   1:  PR[91,3] = PR[90,3] + 57.179;
   1:L PR[91] R[100]mm/sec CNT100;
   1:  PR[91,1] = PR[90,1] + 0.045;
   1:  PR[91,2] = PR[90,2] + -22.058;
   1:  PR[91,3] = PR[90,3] + 57.186;
   1:L PR[91] R[100]mm/sec CNT100;
   1:  PR[91] = PR[90];
   1:  PR[91,1] = PR[90,1] + 1.559;
   1:  PR[91,2] = PR[90,2] + -22.487;
   1:  PR[91,3] = PR[90,3] + 58.520;
   1:L PR[91] R[100]mm/sec CNT100;
   1:  PR[91,1] = PR[90,1] + 2.758;
   1:  PR[91,2] = PR[90,2] + -22.482;
   1:  PR[91,3] = PR[90,3] + 57.203;
   1:L PR[91] R[100]mm/sec CNT100;
   1:  PR[91,1] = PR[90,1] + 3.956;
   1:  PR[91,2] = PR[90,2] + -22.416;
   1:  PR[91,3] = PR[90,3] + 57.213;
   1:L PR[91] R[100]mm/sec CNT100;
   1:  PR[91,1] = PR[90,1] + 5.149;
   1:  PR[91,2] = PR[90,2] + -22.289;
   1:  PR[91,3] = PR[90,3] + 57.223;
   1:L PR[91] R[100]mm/sec CNT100;
   1:  PR[91,1] = PR[90,1] + 6.334;
   1:  PR[91,2] = PR[90,2] + -22.101;
   1:  PR[91,3] = PR[90,3] + 57.234;
   1:L PR[91] R[100]mm/sec CNT100;
   1:  PR[91,1] = PR[90,1] + 7.176;
   1:  PR[91,2] = PR[90,2] + -21.924;
   1:  PR[91,3] = PR[90,3] + 57.244;
   1:L PR[91] R[100]mm/sec CNT100;
   1:  PR[91,1] = PR[90,1] + 7.504;
   1:  PR[91,2] = PR[90,2] + -21.853;
   1:  PR[91,3] = PR[90,3] + 57.252;
   1:L PR[91] R[100]mm/sec CNT100;
   1:  PR[91,1] = PR[90,1] + 8.663;
   1:  PR[91,2] = PR[90,2] + -21.545;
   1:  PR[91,3] = PR[90,3] + 57.255;
   1:L PR[91] R[100]mm/sec CNT100;
   1:  PR[91,1] = PR[90,1] + 9.802;
   1:  PR[91,2] = PR[90,2] + -21.178;
   1:  PR[91,3] = PR[90,3] + 57.265;
   1:L PR[91] R[100]mm/sec CNT100;
   1:  PR[91,1] = PR[90,1] + 10.920;
   1:  PR[91,2] = PR[90,2] + -20.755;
   1:  PR[91,3] = PR[90,3] + 57.275;
   1:L PR[91] R[100]mm/sec CNT100;
   1:  PR[91,1] = PR[90,1] + 12.013;
   1:  PR[91,2] = PR[90,2] + -20.275;
   1:  PR[91,3] = PR[90,3] + 57.286;
   1:L PR[91] R[100]mm/sec CNT100;
   1:  PR[91,1] = PR[90,1] + 13.080;
   1:  PR[91,2] = PR[90,2] + -19.740;
   1:  PR[91,3] = PR[90,3] + 57.296;
   1:L PR[91] R[100]mm/sec CNT100;
   1:  PR[91,1] = PR[90,1] + 14.117;
   1:  PR[91,2] = PR[90,2] + -19.152;
   1:  PR[91,3] = PR[90,3] + 57.306;
   1:L PR[91] R[100]mm/sec CNT100;
   1:  PR[91,1] = PR[90,1] + 14.721;
   1:  PR[91,2] = PR[90,2] + -18.769;
   1:  PR[91,3] = PR[90,3] + 57.317;
   1:L PR[91] R[100]mm/sec CNT100;
   1:  PR[91,1] = PR[90,1] + 15.120;
   1:  PR[91,2] = PR[90,2] + -18.514;
   1:  PR[91,3] = PR[90,3] + 57.323;
   1:L PR[91] R[100]mm/sec CNT100;
   1:  PR[91,1] = PR[90,1] + 16.090;
   1:  PR[91,2] = PR[90,2] + -17.825;
   1:  PR[91,3] = PR[90,3] + 57.327;
   1:L PR[91] R[100]mm/sec CNT100;
   1:  PR[91,1] = PR[90,1] + 17.021;
   1:  PR[91,2] = PR[90,2] + -17.088;
   1:  PR[91,3] = PR[90,3] + 57.337;
   1:L PR[91] R[100]mm/sec CNT100;
   1:  PR[91,1] = PR[90,1] + 17.913;
   1:  PR[91,2] = PR[90,2] + -16.306;
   1:  PR[91,3] = PR[90,3] + 57.348;
   1:L PR[91] R[100]mm/sec CNT100;
   1:  PR[91,1] = PR[90,1] + 18.761;
   1:  PR[91,2] = PR[90,2] + -15.480;
   1:  PR[91,3] = PR[90,3] + 57.358;
   1:L PR[91] R[100]mm/sec CNT100;
   1:  PR[91,1] = PR[90,1] + 19.566;
   1:  PR[91,2] = PR[90,2] + -14.612;
   1:  PR[91,3] = PR[90,3] + 57.368;
   1:L PR[91] R[100]mm/sec CNT100;
   1:  PR[91,1] = PR[90,1] + 20.324;
   1:  PR[91,2] = PR[90,2] + -13.706;
   1:  PR[91,3] = PR[90,3] + 57.378;
   1:L PR[91] R[100]mm/sec CNT100;
   1:  PR[91,1] = PR[90,1] + 21.034;
   1:  PR[91,2] = PR[90,2] + -12.762;
   1:  PR[91,3] = PR[90,3] + 57.389;
   1:L PR[91] R[100]mm/sec CNT100;
   1:  PR[91,1] = PR[90,1] + 21.694;
   1:  PR[91,2] = PR[90,2] + -11.785;
   1:  PR[91,3] = PR[90,3] + 57.399;
   1:L PR[91] R[100]mm/sec CNT100;
   1:  PR[91,1] = PR[90,1] + 22.301;
   1:  PR[91,2] = PR[90,2] + -10.776;
   1:  PR[91,3] = PR[90,3] + 57.409;
   1:L PR[91] R[100]mm/sec CNT100;
   1:  PR[91,1] = PR[90,1] + 22.856;
   1:  PR[91,2] = PR[90,2] + -9.738;
   1:  PR[91,3] = PR[90,3] + 57.419;
   1:L PR[91] R[100]mm/sec CNT100;
   1:  PR[91,1] = PR[90,1] + 23.356;
   1:  PR[91,2] = PR[90,2] + -8.675;
   1:  PR[91,3] = PR[90,3] + 57.429;
   1:L PR[91] R[100]mm/sec CNT100;
   1:  PR[91,1] = PR[90,1] + 23.800;
   1:  PR[91,2] = PR[90,2] + -7.590;
   1:  PR[91,3] = PR[90,3] + 57.440;
   1:L PR[91] R[100]mm/sec CNT100;
   1:  PR[91,1] = PR[90,1] + 24.187;
   1:  PR[91,2] = PR[90,2] + -6.485;
   1:  PR[91,3] = PR[90,3] + 57.450;
   1:L PR[91] R[100]mm/sec CNT100;
   1:  PR[91,1] = PR[90,1] + 24.516;
   1:  PR[91,2] = PR[90,2] + -5.362;
   1:  PR[91,3] = PR[90,3] + 57.460;
   1:L PR[91] R[100]mm/sec CNT100;
   1:  PR[91,1] = PR[90,1] + 24.786;
   1:  PR[91,2] = PR[90,2] + -4.225;
   1:  PR[91,3] = PR[90,3] + 57.470;
   1:L PR[91] R[100]mm/sec CNT100;
   1:  PR[91,1] = PR[90,1] + 24.997;
   1:  PR[91,2] = PR[90,2] + -3.075;
   1:  PR[91,3] = PR[90,3] + 57.480;
   1:L PR[91] R[100]mm/sec CNT100;
   1:  PR[91,1] = PR[90,1] + 25.148;
   1:  PR[91,2] = PR[90,2] + -1.915;
   1:  PR[91,3] = PR[90,3] + 57.490;
   1:L PR[91] R[100]mm/sec CNT100;
   1:  PR[91,1] = PR[90,1] + 25.238;
   1:  PR[91,2] = PR[90,2] + -0.746;
   1:  PR[91,3] = PR[90,3] + 57.500;
   1:L PR[91] R[100]mm/sec CNT100;
   1:  PR[91,1] = PR[90,1] + 25.269;
   1:  PR[91,2] = PR[90,2] + 0.428;
   1:  PR[91,3] = PR[90,3] + 57.510;
   1:L PR[91] R[100]mm/sec CNT100;
   1:  PR[91,1] = PR[90,1] + 25.238;
   1:  PR[91,2] = PR[90,2] + 1.601;
   1:  PR[91,3] = PR[90,3] + 57.521;
   1:L PR[91] R[100]mm/sec CNT100;
   1:  PR[91,1] = PR[90,1] + 25.148;
   1:  PR[91,2] = PR[90,2] + 2.770;
   1:  PR[91,3] = PR[90,3] + 57.531;
   1:L PR[91] R[100]mm/sec CNT100;
   1:  PR[91,1] = PR[90,1] + 24.997;
   1:  PR[91,2] = PR[90,2] + 3.930;
   1:  PR[91,3] = PR[90,3] + 57.541;
   1:L PR[91] R[100]mm/sec CNT100;
   1:  PR[91,1] = PR[90,1] + 24.786;
   1:  PR[91,2] = PR[90,2] + 5.080;
   1:  PR[91,3] = PR[90,3] + 57.551;
   1:L PR[91] R[100]mm/sec CNT100;
   1:  PR[91,1] = PR[90,1] + 24.516;
   1:  PR[91,2] = PR[90,2] + 6.217;
   1:  PR[91,3] = PR[90,3] + 57.561;
   1:L PR[91] R[100]mm/sec CNT100;
   1:  PR[91,1] = PR[90,1] + 24.187;
   1:  PR[91,2] = PR[90,2] + 7.339;
   1:  PR[91,3] = PR[90,3] + 57.571;
   1:L PR[91] R[100]mm/sec CNT100;
   1:  PR[91,1] = PR[90,1] + 23.800;
   1:  PR[91,2] = PR[90,2] + 8.445;
   1:  PR[91,3] = PR[90,3] + 57.581;
   1:L PR[91] R[100]mm/sec CNT100;
   1:  PR[91,1] = PR[90,1] + 23.356;
   1:  PR[91,2] = PR[90,2] + 9.530;
   1:  PR[91,3] = PR[90,3] + 57.592;
   1:L PR[91] R[100]mm/sec CNT100;
   1:  PR[91,1] = PR[90,1] + 22.856;
   1:  PR[91,2] = PR[90,2] + 10.593;
   1:  PR[91,3] = PR[90,3] + 57.602;
   1:L PR[91] R[100]mm/sec CNT100;
   1:  PR[91,1] = PR[90,1] + 22.302;
   1:  PR[91,2] = PR[90,2] + 11.630;
   1:  PR[91,3] = PR[90,3] + 57.612;
   1:L PR[91] R[100]mm/sec CNT100;
   1:  PR[91,1] = PR[90,1] + 21.694;
   1:  PR[91,2] = PR[90,2] + 12.639;
   1:  PR[91,3] = PR[90,3] + 57.622;
   1:L PR[91] R[100]mm/sec CNT100;
   1:  PR[91,1] = PR[90,1] + 21.034;
   1:  PR[91,2] = PR[90,2] + 13.617;
   1:  PR[91,3] = PR[90,3] + 57.632;
   1:L PR[91] R[100]mm/sec CNT100;
   1:  PR[91,1] = PR[90,1] + 20.325;
   1:  PR[91,2] = PR[90,2] + 14.560;
   1:  PR[91,3] = PR[90,3] + 57.642;
   1:L PR[91] R[100]mm/sec CNT100;
   1:  PR[91,1] = PR[90,1] + 19.567;
   1:  PR[91,2] = PR[90,2] + 15.467;
   1:  PR[91,3] = PR[90,3] + 57.653;
   1:L PR[91] R[100]mm/sec CNT100;
   1:  PR[91,1] = PR[90,1] + 18.762;
   1:  PR[91,2] = PR[90,2] + 16.335;
   1:  PR[91,3] = PR[90,3] + 57.663;
   1:L PR[91] R[100]mm/sec CNT100;
   1:  PR[91,1] = PR[90,1] + 17.913;
   1:  PR[91,2] = PR[90,2] + 17.161;
   1:  PR[91,3] = PR[90,3] + 57.673;
   1:L PR[91] R[100]mm/sec CNT100;
   1:  PR[91,1] = PR[90,1] + 17.021;
   1:  PR[91,2] = PR[90,2] + 17.943;
   1:  PR[91,3] = PR[90,3] + 57.683;
   1:L PR[91] R[100]mm/sec CNT100;
   1:  PR[91,1] = PR[90,1] + 16.090;
   1:  PR[91,2] = PR[90,2] + 18.680;
   1:  PR[91,3] = PR[90,3] + 57.694;
   1:L PR[91] R[100]mm/sec CNT100;
   1:  PR[91,1] = PR[90,1] + 15.121;
   1:  PR[91,2] = PR[90,2] + 19.369;
   1:  PR[91,3] = PR[90,3] + 57.704;
   1:L PR[91] R[100]mm/sec CNT100;
   1:  PR[91,1] = PR[90,1] + 14.117;
   1:  PR[91,2] = PR[90,2] + 20.008;
   1:  PR[91,3] = PR[90,3] + 57.714;
   1:L PR[91] R[100]mm/sec CNT100;
   1:  PR[91,1] = PR[90,1] + 13.080;
   1:  PR[91,2] = PR[90,2] + 20.595;
   1:  PR[91,3] = PR[90,3] + 57.725;
   1:L PR[91] R[100]mm/sec CNT100;
   1:  PR[91,1] = PR[90,1] + 12.013;
   1:  PR[91,2] = PR[90,2] + 21.130;
   1:  PR[91,3] = PR[90,3] + 57.735;
   1:L PR[91] R[100]mm/sec CNT100;
   1:  PR[91,1] = PR[90,1] + 10.919;
   1:  PR[91,2] = PR[90,2] + 21.610;
   1:  PR[91,3] = PR[90,3] + 57.745;
   1:L PR[91] R[100]mm/sec CNT100;
   1:  PR[91,1] = PR[90,1] + 9.802;
   1:  PR[91,2] = PR[90,2] + 22.033;
   1:  PR[91,3] = PR[90,3] + 57.756;
   1:L PR[91] R[100]mm/sec CNT100;
   1:  PR[91,1] = PR[90,1] + 8.662;
   1:  PR[91,2] = PR[90,2] + 22.400;
   1:  PR[91,3] = PR[90,3] + 57.766;
   1:L PR[91] R[100]mm/sec CNT100;
   1:  PR[91,1] = PR[90,1] + 7.503;
   1:  PR[91,2] = PR[90,2] + 22.708;
   1:  PR[91,3] = PR[90,3] + 57.776;
   1:L PR[91] R[100]mm/sec CNT100;
   1:  PR[91,1] = PR[90,1] + 7.175;
   1:  PR[91,2] = PR[90,2] + 22.780;
   1:  PR[91,3] = PR[90,3] + 57.787;
   1:L PR[91] R[100]mm/sec CNT100;
   1:  PR[91,1] = PR[90,1] + 6.333;
   1:  PR[91,2] = PR[90,2] + 22.956;
   1:  PR[91,3] = PR[90,3] + 57.790;
   1:L PR[91] R[100]mm/sec CNT100;
   1:  PR[91,1] = PR[90,1] + 5.148;
   1:  PR[91,2] = PR[90,2] + 23.144;
   1:  PR[91,3] = PR[90,3] + 57.797;
   1:L PR[91] R[100]mm/sec CNT100;
   1:  PR[91,1] = PR[90,1] + 3.955;
   1:  PR[91,2] = PR[90,2] + 23.271;
   1:  PR[91,3] = PR[90,3] + 57.807;
   1:L PR[91] R[100]mm/sec CNT100;
   1:  PR[91,1] = PR[90,1] + 2.757;
   1:  PR[91,2] = PR[90,2] + 23.337;
   1:  PR[91,3] = PR[90,3] + 57.818;
   1:L PR[91] R[100]mm/sec CNT100;
   1:  PR[91,1] = PR[90,1] + 1.557;
   1:  PR[91,2] = PR[90,2] + 23.342;
   1:  PR[91,3] = PR[90,3] + 57.828;
   1:L PR[91] R[100]mm/sec CNT100;
   1:  PR[91,1] = PR[90,1] + 0.088;
   1:  PR[91,2] = PR[90,2] + 23.262;
   1:  PR[91,3] = PR[90,3] + 57.839;
   1:L PR[91] R[100]mm/sec CNT100;
   1:  PR[91,1] = PR[90,1] + -0.337;
   1:  PR[91,3] = PR[90,3] + 57.851;
   1:L PR[91] R[100]mm/sec CNT100;
   1:  PR[91,1] = PR[90,1] + -1.797;
   1:  PR[91,2] = PR[90,2] + 23.342;
   1:  PR[91,3] = PR[90,3] + 57.855;
   1:L PR[91] R[100]mm/sec CNT100;
   1:  PR[91,1] = PR[90,1] + -2.726;
   1:  PR[91,2] = PR[90,2] + 23.340;
   1:  PR[91,3] = PR[90,3] + 57.868;
   1:L PR[91] R[100]mm/sec CNT100;
   1:  PR[91,1] = PR[90,1] + -4.196;
   1:  PR[91,2] = PR[90,2] + 23.271;
   1:  PR[91,3] = PR[90,3] + 57.876;
   1:L PR[91] R[100]mm/sec CNT100;
   1:  PR[91,1] = PR[90,1] + -5.387;
   1:  PR[91,2] = PR[90,2] + 23.144;
   1:  PR[91,3] = PR[90,3] + 57.888;
   1:L PR[91] R[100]mm/sec CNT100;
   1:  PR[91,1] = PR[90,1] + -6.572;
   1:  PR[91,2] = PR[90,2] + 22.956;
   1:  PR[91,3] = PR[90,3] + 57.899;
   1:L PR[91] R[100]mm/sec CNT100;
   1:  PR[91,1] = PR[90,1] + -7.413;
   1:  PR[91,2] = PR[90,2] + 22.780;
   1:  PR[91,3] = PR[90,3] + 57.909;
   1:L PR[91] R[100]mm/sec CNT100;
   1:  PR[91,1] = PR[90,1] + -7.742;
   1:  PR[91,2] = PR[90,2] + 22.708;
   1:  PR[91,3] = PR[90,3] + 57.917;
   1:L PR[91] R[100]mm/sec CNT100;
   1:  PR[91,1] = PR[90,1] + -8.901;
   1:  PR[91,2] = PR[90,2] + 22.400;
   1:  PR[91,3] = PR[90,3] + 57.920;
   1:L PR[91] R[100]mm/sec CNT100;
   1:  PR[91,1] = PR[90,1] + -10.040;
   1:  PR[91,2] = PR[90,2] + 22.034;
   1:  PR[91,3] = PR[90,3] + 57.930;
   1:L PR[91] R[100]mm/sec CNT100;
   1:  PR[91,1] = PR[90,1] + -11.158;
   1:  PR[91,2] = PR[90,2] + 21.610;
   1:  PR[91,3] = PR[90,3] + 57.940;
   1:L PR[91] R[100]mm/sec CNT100;
   1:  PR[91,1] = PR[90,1] + -12.251;
   1:  PR[91,2] = PR[90,2] + 21.130;
   1:  PR[91,3] = PR[90,3] + 57.951;
   1:L PR[91] R[100]mm/sec CNT100;
   1:  PR[91,1] = PR[90,1] + -13.318;
   1:  PR[91,2] = PR[90,2] + 20.595;
   1:  PR[91,3] = PR[90,3] + 57.961;
   1:L PR[91] R[100]mm/sec CNT100;
   1:  PR[91,1] = PR[90,1] + -14.355;
   1:  PR[91,2] = PR[90,2] + 20.008;
   1:  PR[91,3] = PR[90,3] + 57.971;
   1:L PR[91] R[100]mm/sec CNT100;
   1:  PR[91,1] = PR[90,1] + -15.359;
   1:  PR[91,2] = PR[90,2] + 19.368;
   1:  PR[91,3] = PR[90,3] + 57.982;
   1:L PR[91] R[100]mm/sec CNT100;
   1:  PR[91,1] = PR[90,1] + -16.329;
   1:  PR[91,2] = PR[90,2] + 18.679;
   1:  PR[91,3] = PR[90,3] + 57.992;
   1:L PR[91] R[100]mm/sec CNT100;
   1:  PR[91,1] = PR[90,1] + -17.260;
   1:  PR[91,2] = PR[90,2] + 17.943;
   1:  PR[91,3] = PR[90,3] + 58.002;
   1:L PR[91] R[100]mm/sec CNT100;
   1:  PR[91,1] = PR[90,1] + -18.151;
   1:  PR[91,2] = PR[90,2] + 17.161;
   1:  PR[91,3] = PR[90,3] + 58.013;
   1:L PR[91] R[100]mm/sec CNT100;
   1:  PR[91,1] = PR[90,1] + -19.000;
   1:  PR[91,2] = PR[90,2] + 16.335;
   1:  PR[91,3] = PR[90,3] + 58.023;
   1:L PR[91] R[100]mm/sec CNT100;
   1:  PR[91,1] = PR[90,1] + -19.805;
   1:  PR[91,2] = PR[90,2] + 15.467;
   1:  PR[91,3] = PR[90,3] + 58.033;
   1:L PR[91] R[100]mm/sec CNT100;
   1:  PR[91,1] = PR[90,1] + -20.563;
   1:  PR[91,2] = PR[90,2] + 14.561;
   1:  PR[91,3] = PR[90,3] + 58.043;
   1:L PR[91] R[100]mm/sec CNT100;
   1:  PR[91,1] = PR[90,1] + -21.273;
   1:  PR[91,2] = PR[90,2] + 13.618;
   1:  PR[91,3] = PR[90,3] + 58.054;
   1:L PR[91] R[100]mm/sec CNT100;
   1:  PR[91,1] = PR[90,1] + -21.933;
   1:  PR[91,2] = PR[90,2] + 12.640;
   1:  PR[91,3] = PR[90,3] + 58.064;
   1:L PR[91] R[100]mm/sec CNT100;
   1:  PR[91,1] = PR[90,1] + -22.540;
   1:  PR[91,2] = PR[90,2] + 11.631;
   1:  PR[91,3] = PR[90,3] + 58.074;
   1:L PR[91] R[100]mm/sec CNT100;
   1:  PR[91,1] = PR[90,1] + -23.095;
   1:  PR[91,2] = PR[90,2] + 10.593;
   1:  PR[91,3] = PR[90,3] + 58.084;
   1:L PR[91] R[100]mm/sec CNT100;
   1:  PR[91,1] = PR[90,1] + -23.594;
   1:  PR[91,2] = PR[90,2] + 9.530;
   1:  PR[91,3] = PR[90,3] + 58.094;
   1:L PR[91] R[100]mm/sec CNT100;
   1:  PR[91,1] = PR[90,1] + -24.038;
   1:  PR[91,2] = PR[90,2] + 8.444;
   1:  PR[91,3] = PR[90,3] + 58.105;
   1:L PR[91] R[100]mm/sec CNT100;
   1:  PR[91,1] = PR[90,1] + -24.425;
   1:  PR[91,2] = PR[90,2] + 7.338;
   1:  PR[91,3] = PR[90,3] + 58.115;
   1:L PR[91] R[100]mm/sec CNT100;
   1:  PR[91,1] = PR[90,1] + -24.754;
   1:  PR[91,2] = PR[90,2] + 6.215;
   1:  PR[91,3] = PR[90,3] + 58.125;
   1:L PR[91] R[100]mm/sec CNT100;
   1:  PR[91,1] = PR[90,1] + -25.024;
   1:  PR[91,2] = PR[90,2] + 5.078;
   1:  PR[91,3] = PR[90,3] + 58.135;
   1:L PR[91] R[100]mm/sec CNT100;
   1:  PR[91,1] = PR[90,1] + -25.235;
   1:  PR[91,2] = PR[90,2] + 3.929;
   1:  PR[91,3] = PR[90,3] + 58.145;
   1:L PR[91] R[100]mm/sec CNT100;
   1:  PR[91,1] = PR[90,1] + -25.386;
   1:  PR[91,2] = PR[90,2] + 2.769;
   1:  PR[91,3] = PR[90,3] + 58.155;
   1:L PR[91] R[100]mm/sec CNT100;
   1:  PR[91,1] = PR[90,1] + -25.477;
   1:  PR[91,2] = PR[90,2] + 1.601;
   1:  PR[91,3] = PR[90,3] + 58.165;
   1:L PR[91] R[100]mm/sec CNT100;
   1:  PR[91,1] = PR[90,1] + -25.507;
   1:  PR[91,2] = PR[90,2] + 0.428;
   1:  PR[91,3] = PR[90,3] + 58.175;
   1:L PR[91] R[100]mm/sec CNT100;
   1:  PR[91,1] = PR[90,1] + -25.477;
   1:  PR[91,2] = PR[90,2] + -0.746;
   1:  PR[91,3] = PR[90,3] + 58.186;
   1:L PR[91] R[100]mm/sec CNT100;
   1:  PR[91,1] = PR[90,1] + -25.386;
   1:  PR[91,2] = PR[90,2] + -1.914;
   1:  PR[91,3] = PR[90,3] + 58.196;
   1:L PR[91] R[100]mm/sec CNT100;
   1:  PR[91,1] = PR[90,1] + -25.235;
   1:  PR[91,2] = PR[90,2] + -3.074;
   1:  PR[91,3] = PR[90,3] + 58.206;
   1:L PR[91] R[100]mm/sec CNT100;
   1:  PR[91,1] = PR[90,1] + -25.024;
   1:  PR[91,2] = PR[90,2] + -4.223;
   1:  PR[91,3] = PR[90,3] + 58.216;
   1:L PR[91] R[100]mm/sec CNT100;
   1:  PR[91,1] = PR[90,1] + -24.754;
   1:  PR[91,2] = PR[90,2] + -5.361;
   1:  PR[91,3] = PR[90,3] + 58.226;
   1:L PR[91] R[100]mm/sec CNT100;
   1:  PR[91,1] = PR[90,1] + -24.425;
   1:  PR[91,2] = PR[90,2] + -6.483;
   1:  PR[91,3] = PR[90,3] + 58.236;
   1:L PR[91] R[100]mm/sec CNT100;
   1:  PR[91,1] = PR[90,1] + -24.038;
   1:  PR[91,2] = PR[90,2] + -7.589;
   1:  PR[91,3] = PR[90,3] + 58.246;
   1:L PR[91] R[100]mm/sec CNT100;
   1:  PR[91,1] = PR[90,1] + -23.594;
   1:  PR[91,2] = PR[90,2] + -8.675;
   1:  PR[91,3] = PR[90,3] + 58.257;
   1:L PR[91] R[100]mm/sec CNT100;
   1:  PR[91,1] = PR[90,1] + -23.094;
   1:  PR[91,2] = PR[90,2] + -9.739;
   1:  PR[91,3] = PR[90,3] + 58.267;
   1:L PR[91] R[100]mm/sec CNT100;
   1:  PR[91,1] = PR[90,1] + -22.540;
   1:  PR[91,2] = PR[90,2] + -10.776;
   1:  PR[91,3] = PR[90,3] + 58.277;
   1:L PR[91] R[100]mm/sec CNT100;
   1:  PR[91,1] = PR[90,1] + -21.932;
   1:  PR[91,2] = PR[90,2] + -11.786;
   1:  PR[91,3] = PR[90,3] + 58.287;
   1:L PR[91] R[100]mm/sec CNT100;
   1:  PR[91,1] = PR[90,1] + -21.273;
   1:  PR[91,2] = PR[90,2] + -12.763;
   1:  PR[91,3] = PR[90,3] + 58.297;
   1:L PR[91] R[100]mm/sec CNT100;
   1:  PR[91,1] = PR[90,1] + -20.563;
   1:  PR[91,2] = PR[90,2] + -13.706;
   1:  PR[91,3] = PR[90,3] + 58.307;
   1:L PR[91] R[100]mm/sec CNT100;
   1:  PR[91,1] = PR[90,1] + -19.805;
   1:  PR[91,2] = PR[90,2] + -14.613;
   1:  PR[91,3] = PR[90,3] + 58.318;
   1:L PR[91] R[100]mm/sec CNT100;
   1:  PR[91,1] = PR[90,1] + -19.000;
   1:  PR[91,2] = PR[90,2] + -15.480;
   1:  PR[91,3] = PR[90,3] + 58.328;
   1:L PR[91] R[100]mm/sec CNT100;
   1:  PR[91,1] = PR[90,1] + -18.151;
   1:  PR[91,2] = PR[90,2] + -16.306;
   1:  PR[91,3] = PR[90,3] + 58.338;
   1:L PR[91] R[100]mm/sec CNT100;
   1:  PR[91,1] = PR[90,1] + -17.260;
   1:  PR[91,2] = PR[90,2] + -17.088;
   1:  PR[91,3] = PR[90,3] + 58.348;
   1:L PR[91] R[100]mm/sec CNT100;
   1:  PR[91,1] = PR[90,1] + -16.328;
   1:  PR[91,2] = PR[90,2] + -17.824;
   1:  PR[91,3] = PR[90,3] + 58.359;
   1:L PR[91] R[100]mm/sec CNT100;
   1:  PR[91,1] = PR[90,1] + -15.359;
   1:  PR[91,2] = PR[90,2] + -18.513;
   1:  PR[91,3] = PR[90,3] + 58.369;
   1:L PR[91] R[100]mm/sec CNT100;
   1:  PR[91,1] = PR[90,1] + -14.355;
   1:  PR[91,2] = PR[90,2] + -19.153;
   1:  PR[91,3] = PR[90,3] + 58.379;
   1:L PR[91] R[100]mm/sec CNT100;
   1:  PR[91,1] = PR[90,1] + -13.318;
   1:  PR[91,2] = PR[90,2] + -19.740;
   1:  PR[91,3] = PR[90,3] + 58.390;
   1:L PR[91] R[100]mm/sec CNT100;
   1:  PR[91,1] = PR[90,1] + -12.252;
   1:  PR[91,2] = PR[90,2] + -20.275;
   1:  PR[91,3] = PR[90,3] + 58.400;
   1:L PR[91] R[100]mm/sec CNT100;
   1:  PR[91,1] = PR[90,1] + -11.158;
   1:  PR[91,2] = PR[90,2] + -20.755;
   1:  PR[91,3] = PR[90,3] + 58.410;
   1:L PR[91] R[100]mm/sec CNT100;
   1:  PR[91,1] = PR[90,1] + -10.039;
   1:  PR[91,2] = PR[90,2] + -21.179;
   1:  PR[91,3] = PR[90,3] + 58.421;
   1:L PR[91] R[100]mm/sec CNT100;
   1:  PR[91,1] = PR[90,1] + -9.682;
   1:  PR[91,2] = PR[90,2] + -21.295;
   1:  PR[91,3] = PR[90,3] + 58.431;
   1:L PR[91] R[100]mm/sec CNT100;
   1:  PR[91,1] = PR[90,1] + -8.902;
   1:  PR[91,2] = PR[90,2] + -21.544;
   1:  PR[91,3] = PR[90,3] + 58.434;
   1:L PR[91] R[100]mm/sec CNT100;
   1:  PR[91,1] = PR[90,1] + -7.744;
   1:  PR[91,2] = PR[90,2] + -21.852;
   1:  PR[91,3] = PR[90,3] + 58.441;
   1:L PR[91] R[100]mm/sec CNT100;
   1:  PR[91,1] = PR[90,1] + -6.572;
   1:  PR[91,2] = PR[90,2] + -22.101;
   1:  PR[91,3] = PR[90,3] + 58.452;
   1:L PR[91] R[100]mm/sec CNT100;
   1:  PR[91,1] = PR[90,1] + -5.388;
   1:  PR[91,2] = PR[90,2] + -22.289;
   1:  PR[91,3] = PR[90,3] + 58.462;
   1:L PR[91] R[100]mm/sec CNT100;
   1:  PR[91,1] = PR[90,1] + -4.197;
   1:  PR[91,2] = PR[90,2] + -22.416;
   1:  PR[91,3] = PR[90,3] + 58.472;
   1:L PR[91] R[100]mm/sec CNT100;
   1:  PR[91,1] = PR[90,1] + -2.727;
   1:  PR[91,2] = PR[90,2] + -22.485;
   1:  PR[91,3] = PR[90,3] + 58.483;
   1:L PR[91] R[100]mm/sec CNT100;
   1:  PR[91,1] = PR[90,1] + -1.798;
   1:  PR[91,2] = PR[90,2] + -22.487;
   1:  PR[91,3] = PR[90,3] + 58.496;
   1:L PR[91] R[100]mm/sec CNT100;
   1:  PR[91,1] = PR[90,1] + -0.337;
   1:  PR[91,2] = PR[90,2] + -22.407;
   1:  PR[91,3] = PR[90,3] + 58.504;
   1:L PR[91] R[100]mm/sec CNT100;
   1:  PR[91,1] = PR[90,1] + 0.098;
   1:  PR[91,3] = PR[90,3] + 58.516;
   1:L PR[91] R[100]mm/sec CNT100;
   1:  PR[91] = PR[90];
   1:  PR[91,1] = PR[90,1] + 0.946;
   1:  PR[91,2] = PR[90,2] + -22.790;
   1:  PR[91,3] = PR[90,3] + 59.850;
   1:L PR[91] R[100]mm/sec CNT100;
   1:  PR[91,1] = PR[90,1] + 2.164;
   1:  PR[91,2] = PR[90,2] + -22.792;
   1:  PR[91,3] = PR[90,3] + 58.528;
   1:L PR[91] R[100]mm/sec CNT100;
   1:  PR[91,1] = PR[90,1] + 3.379;
   1:  PR[91,2] = PR[90,2] + -22.731;
   1:  PR[91,3] = PR[90,3] + 58.538;
   1:L PR[91] R[100]mm/sec CNT100;
   1:  PR[91,1] = PR[90,1] + 4.589;
   1:  PR[91,2] = PR[90,2] + -22.607;
   1:  PR[91,3] = PR[90,3] + 58.549;
   1:L PR[91] R[100]mm/sec CNT100;
   1:  PR[91,1] = PR[90,1] + 5.790;
   1:  PR[91,2] = PR[90,2] + -22.422;
   1:  PR[91,3] = PR[90,3] + 58.559;
   1:L PR[91] R[100]mm/sec CNT100;
   1:  PR[91,1] = PR[90,1] + 6.979;
   1:  PR[91,2] = PR[90,2] + -22.175;
   1:  PR[91,3] = PR[90,3] + 58.570;
   1:L PR[91] R[100]mm/sec CNT100;
   1:  PR[91,1] = PR[90,1] + 8.153;
   1:  PR[91,2] = PR[90,2] + -21.867;
   1:  PR[91,3] = PR[90,3] + 58.580;
   1:L PR[91] R[100]mm/sec CNT100;
   1:  PR[91,1] = PR[90,1] + 9.308;
   1:  PR[91,2] = PR[90,2] + -21.500;
   1:  PR[91,3] = PR[90,3] + 58.591;
   1:L PR[91] R[100]mm/sec CNT100;
   1:  PR[91,1] = PR[90,1] + 10.625;
   1:  PR[91,2] = PR[90,2] + -20.997;
   1:  PR[91,3] = PR[90,3] + 58.602;
   1:L PR[91] R[100]mm/sec CNT100;
   1:  PR[91,1] = PR[90,1] + 11.554;
   1:  PR[91,2] = PR[90,2] + -20.591;
   1:  PR[91,3] = PR[90,3] + 58.614;
   1:L PR[91] R[100]mm/sec CNT100;
   1:  PR[91,1] = PR[90,1] + 12.638;
   1:  PR[91,2] = PR[90,2] + -20.051;
   1:  PR[91,3] = PR[90,3] + 58.623;
   1:L PR[91] R[100]mm/sec CNT100;
   1:  PR[91,1] = PR[90,1] + 13.691;
   1:  PR[91,2] = PR[90,2] + -19.458;
   1:  PR[91,3] = PR[90,3] + 58.633;
   1:L PR[91] R[100]mm/sec CNT100;
   1:  PR[91,1] = PR[90,1] + 14.711;
   1:  PR[91,2] = PR[90,2] + -18.812;
   1:  PR[91,3] = PR[90,3] + 58.643;
   1:L PR[91] R[100]mm/sec CNT100;
   1:  PR[91,1] = PR[90,1] + 15.696;
   1:  PR[91,2] = PR[90,2] + -18.115;
   1:  PR[91,3] = PR[90,3] + 58.654;
   1:L PR[91] R[100]mm/sec CNT100;
   1:  PR[91,1] = PR[90,1] + 16.643;
   1:  PR[91,2] = PR[90,2] + -17.369;
   1:  PR[91,3] = PR[90,3] + 58.664;
   1:L PR[91] R[100]mm/sec CNT100;
   1:  PR[91,1] = PR[90,1] + 17.549;
   1:  PR[91,2] = PR[90,2] + -16.576;
   1:  PR[91,3] = PR[90,3] + 58.675;
   1:L PR[91] R[100]mm/sec CNT100;
   1:  PR[91,1] = PR[90,1] + 18.412;
   1:  PR[91,2] = PR[90,2] + -15.739;
   1:  PR[91,3] = PR[90,3] + 58.685;
   1:L PR[91] R[100]mm/sec CNT100;
   1:  PR[91,1] = PR[90,1] + 19.230;
   1:  PR[91,2] = PR[90,2] + -14.859;
   1:  PR[91,3] = PR[90,3] + 58.696;
   1:L PR[91] R[100]mm/sec CNT100;
   1:  PR[91,1] = PR[90,1] + 20.001;
   1:  PR[91,2] = PR[90,2] + -13.939;
   1:  PR[91,3] = PR[90,3] + 58.706;
   1:L PR[91] R[100]mm/sec CNT100;
   1:  PR[91,1] = PR[90,1] + 20.723;
   1:  PR[91,2] = PR[90,2] + -12.982;
   1:  PR[91,3] = PR[90,3] + 58.717;
   1:L PR[91] R[100]mm/sec CNT100;
   1:  PR[91,1] = PR[90,1] + 21.404;
   1:  PR[91,2] = PR[90,2] + -11.972;
   1:  PR[91,3] = PR[90,3] + 58.727;
   1:L PR[91] R[100]mm/sec CNT100;
   1:  PR[91,1] = PR[90,1] + 22.016;
   1:  PR[91,2] = PR[90,2] + -10.957;
   1:  PR[91,3] = PR[90,3] + 58.738;
   1:L PR[91] R[100]mm/sec CNT100;
   1:  PR[91,1] = PR[90,1] + 22.576;
   1:  PR[91,2] = PR[90,2] + -9.911;
   1:  PR[91,3] = PR[90,3] + 58.748;
   1:L PR[91] R[100]mm/sec CNT100;
   1:  PR[91,1] = PR[90,1] + 23.085;
   1:  PR[91,2] = PR[90,2] + -8.830;
   1:  PR[91,3] = PR[90,3] + 58.758;
   1:L PR[91] R[100]mm/sec CNT100;
   1:  PR[91,1] = PR[90,1] + 23.537;
   1:  PR[91,2] = PR[90,2] + -7.727;
   1:  PR[91,3] = PR[90,3] + 58.768;
   1:L PR[91] R[100]mm/sec CNT100;
   1:  PR[91,1] = PR[90,1] + 23.931;
   1:  PR[91,2] = PR[90,2] + -6.602;
   1:  PR[91,3] = PR[90,3] + 58.779;
   1:L PR[91] R[100]mm/sec CNT100;
   1:  PR[91,1] = PR[90,1] + 24.266;
   1:  PR[91,2] = PR[90,2] + -5.460;
   1:  PR[91,3] = PR[90,3] + 58.789;
   1:L PR[91] R[100]mm/sec CNT100;
   1:  PR[91,1] = PR[90,1] + 24.541;
   1:  PR[91,2] = PR[90,2] + -4.303;
   1:  PR[91,3] = PR[90,3] + 58.799;
   1:L PR[91] R[100]mm/sec CNT100;
   1:  PR[91,1] = PR[90,1] + 24.756;
   1:  PR[91,2] = PR[90,2] + -3.132;
   1:  PR[91,3] = PR[90,3] + 58.810;
   1:L PR[91] R[100]mm/sec CNT100;
   1:  PR[91,1] = PR[90,1] + 24.909;
   1:  PR[91,2] = PR[90,2] + -1.952;
   1:  PR[91,3] = PR[90,3] + 58.820;
   1:L PR[91] R[100]mm/sec CNT100;
   1:  PR[91,1] = PR[90,1] + 25.002;
   1:  PR[91,2] = PR[90,2] + -0.765;
   1:  PR[91,3] = PR[90,3] + 58.830;
   1:L PR[91] R[100]mm/sec CNT100;
   1:  PR[91,1] = PR[90,1] + 25.033;
   1:  PR[91,2] = PR[90,2] + 0.428;
   1:  PR[91,3] = PR[90,3] + 58.841;
   1:L PR[91] R[100]mm/sec CNT100;
   1:  PR[91,1] = PR[90,1] + 25.002;
   1:  PR[91,2] = PR[90,2] + 1.620;
   1:  PR[91,3] = PR[90,3] + 58.851;
   1:L PR[91] R[100]mm/sec CNT100;
   1:  PR[91,1] = PR[90,1] + 24.909;
   1:  PR[91,2] = PR[90,2] + 2.808;
   1:  PR[91,3] = PR[90,3] + 58.861;
   1:L PR[91] R[100]mm/sec CNT100;
   1:  PR[91,1] = PR[90,1] + 24.755;
   1:  PR[91,2] = PR[90,2] + 3.988;
   1:  PR[91,3] = PR[90,3] + 58.872;
   1:L PR[91] R[100]mm/sec CNT100;
   1:  PR[91,1] = PR[90,1] + 24.541;
   1:  PR[91,2] = PR[90,2] + 5.158;
   1:  PR[91,3] = PR[90,3] + 58.882;
   1:L PR[91] R[100]mm/sec CNT100;
   1:  PR[91,1] = PR[90,1] + 24.266;
   1:  PR[91,2] = PR[90,2] + 6.316;
   1:  PR[91,3] = PR[90,3] + 58.892;
   1:L PR[91] R[100]mm/sec CNT100;
   1:  PR[91,1] = PR[90,1] + 23.930;
   1:  PR[91,2] = PR[90,2] + 7.458;
   1:  PR[91,3] = PR[90,3] + 58.903;
   1:L PR[91] R[100]mm/sec CNT100;
   1:  PR[91,1] = PR[90,1] + 23.530;
   1:  PR[91,2] = PR[90,2] + 8.598;
   1:  PR[91,3] = PR[90,3] + 58.913;
   1:L PR[91] R[100]mm/sec CNT100;
   1:  PR[91,1] = PR[90,1] + 23.081;
   1:  PR[91,2] = PR[90,2] + 9.695;
   1:  PR[91,3] = PR[90,3] + 58.923;
   1:L PR[91] R[100]mm/sec CNT100;
   1:  PR[91,1] = PR[90,1] + 22.575;
   1:  PR[91,2] = PR[90,2] + 10.767;
   1:  PR[91,3] = PR[90,3] + 58.934;
   1:L PR[91] R[100]mm/sec CNT100;
   1:  PR[91,1] = PR[90,1] + 22.012;
   1:  PR[91,2] = PR[90,2] + 11.821;
   1:  PR[91,3] = PR[90,3] + 58.944;
   1:L PR[91] R[100]mm/sec CNT100;
   1:  PR[91,1] = PR[90,1] + 21.393;
   1:  PR[91,2] = PR[90,2] + 12.845;
   1:  PR[91,3] = PR[90,3] + 58.954;
   1:L PR[91] R[100]mm/sec CNT100;
   1:  PR[91,1] = PR[90,1] + 20.722;
   1:  PR[91,2] = PR[90,2] + 13.838;
   1:  PR[91,3] = PR[90,3] + 58.965;
   1:L PR[91] R[100]mm/sec CNT100;
   1:  PR[91,1] = PR[90,1] + 20.000;
   1:  PR[91,2] = PR[90,2] + 14.795;
   1:  PR[91,3] = PR[90,3] + 58.975;
   1:L PR[91] R[100]mm/sec CNT100;
   1:  PR[91,1] = PR[90,1] + 19.229;
   1:  PR[91,2] = PR[90,2] + 15.715;
   1:  PR[91,3] = PR[90,3] + 58.986;
   1:L PR[91] R[100]mm/sec CNT100;
   1:  PR[91,1] = PR[90,1] + 18.411;
   1:  PR[91,2] = PR[90,2] + 16.595;
   1:  PR[91,3] = PR[90,3] + 58.996;
   1:L PR[91] R[100]mm/sec CNT100;
   1:  PR[91,1] = PR[90,1] + 17.547;
   1:  PR[91,2] = PR[90,2] + 17.432;
   1:  PR[91,3] = PR[90,3] + 59.006;
   1:L PR[91] R[100]mm/sec CNT100;
   1:  PR[91,1] = PR[90,1] + 16.641;
   1:  PR[91,2] = PR[90,2] + 18.225;
   1:  PR[91,3] = PR[90,3] + 59.017;
   1:L PR[91] R[100]mm/sec CNT100;
   1:  PR[91,1] = PR[90,1] + 15.694;
   1:  PR[91,2] = PR[90,2] + 18.971;
   1:  PR[91,3] = PR[90,3] + 59.027;
   1:L PR[91] R[100]mm/sec CNT100;
   1:  PR[91,1] = PR[90,1] + 14.710;
   1:  PR[91,2] = PR[90,2] + 19.668;
   1:  PR[91,3] = PR[90,3] + 59.038;
   1:L PR[91] R[100]mm/sec CNT100;
   1:  PR[91,1] = PR[90,1] + 13.689;
   1:  PR[91,2] = PR[90,2] + 20.314;
   1:  PR[91,3] = PR[90,3] + 59.048;
   1:L PR[91] R[100]mm/sec CNT100;
   1:  PR[91,1] = PR[90,1] + 12.636;
   1:  PR[91,2] = PR[90,2] + 20.908;
   1:  PR[91,3] = PR[90,3] + 59.059;
   1:L PR[91] R[100]mm/sec CNT100;
   1:  PR[91,1] = PR[90,1] + 11.553;
   1:  PR[91,2] = PR[90,2] + 21.447;
   1:  PR[91,3] = PR[90,3] + 59.069;
   1:L PR[91] R[100]mm/sec CNT100;
   1:  PR[91,1] = PR[90,1] + 10.442;
   1:  PR[91,2] = PR[90,2] + 21.930;
   1:  PR[91,3] = PR[90,3] + 59.080;
   1:L PR[91] R[100]mm/sec CNT100;
   1:  PR[91,1] = PR[90,1] + 9.307;
   1:  PR[91,2] = PR[90,2] + 22.356;
   1:  PR[91,3] = PR[90,3] + 59.090;
   1:L PR[91] R[100]mm/sec CNT100;
   1:  PR[91,1] = PR[90,1] + 8.151;
   1:  PR[91,2] = PR[90,2] + 22.723;
   1:  PR[91,3] = PR[90,3] + 59.101;
   1:L PR[91] R[100]mm/sec CNT100;
   1:  PR[91,1] = PR[90,1] + 6.977;
   1:  PR[91,2] = PR[90,2] + 23.030;
   1:  PR[91,3] = PR[90,3] + 59.111;
   1:L PR[91] R[100]mm/sec CNT100;
   1:  PR[91,1] = PR[90,1] + 5.788;
   1:  PR[91,2] = PR[90,2] + 23.277;
   1:  PR[91,3] = PR[90,3] + 59.122;
   1:L PR[91] R[100]mm/sec CNT100;
   1:  PR[91,1] = PR[90,1] + 4.586;
   1:  PR[91,2] = PR[90,2] + 23.463;
   1:  PR[91,3] = PR[90,3] + 59.132;
   1:L PR[91] R[100]mm/sec CNT100;
   1:  PR[91,1] = PR[90,1] + 3.377;
   1:  PR[91,2] = PR[90,2] + 23.586;
   1:  PR[91,3] = PR[90,3] + 59.143;
   1:L PR[91] R[100]mm/sec CNT100;
   1:  PR[91,1] = PR[90,1] + 2.162;
   1:  PR[91,2] = PR[90,2] + 23.647;
   1:  PR[91,3] = PR[90,3] + 59.153;
   1:L PR[91] R[100]mm/sec CNT100;
   1:  PR[91,1] = PR[90,1] + 0.943;
   1:  PR[91,2] = PR[90,2] + 23.646;
   1:  PR[91,3] = PR[90,3] + 59.164;
   1:L PR[91] R[100]mm/sec CNT100;
   1:  PR[91,1] = PR[90,1] + 0.051;
   1:  PR[91,2] = PR[90,2] + 23.602;
   1:  PR[91,3] = PR[90,3] + 59.174;
   1:L PR[91] R[100]mm/sec CNT100;
   1:  PR[91,1] = PR[90,1] + -0.290;
   1:  PR[91,3] = PR[90,3] + 59.182;
   1:L PR[91] R[100]mm/sec CNT100;
   1:  PR[91,1] = PR[90,1] + -1.181;
   1:  PR[91,2] = PR[90,2] + 23.646;
   1:  PR[91,3] = PR[90,3] + 59.185;
   1:L PR[91] R[100]mm/sec CNT100;
   1:  PR[91,1] = PR[90,1] + -2.400;
   1:  PR[91,2] = PR[90,2] + 23.647;
   1:  PR[91,3] = PR[90,3] + 59.193;
   1:L PR[91] R[100]mm/sec CNT100;
   1:  PR[91,1] = PR[90,1] + -3.615;
   1:  PR[91,2] = PR[90,2] + 23.586;
   1:  PR[91,3] = PR[90,3] + 59.203;
   1:L PR[91] R[100]mm/sec CNT100;
   1:  PR[91,1] = PR[90,1] + -4.823;
   1:  PR[91,2] = PR[90,2] + 23.463;
   1:  PR[91,3] = PR[90,3] + 59.214;
   1:L PR[91] R[100]mm/sec CNT100;
   1:  PR[91,1] = PR[90,1] + -6.286;
   1:  PR[91,2] = PR[90,2] + 23.226;
   1:  PR[91,3] = PR[90,3] + 59.224;
   1:L PR[91] R[100]mm/sec CNT100;
   1:  PR[91,1] = PR[90,1] + -7.215;
   1:  PR[91,2] = PR[90,2] + 23.031;
   1:  PR[91,3] = PR[90,3] + 59.237;
   1:L PR[91] R[100]mm/sec CNT100;
   1:  PR[91,1] = PR[90,1] + -8.390;
   1:  PR[91,2] = PR[90,2] + 22.723;
   1:  PR[91,3] = PR[90,3] + 59.245;
   1:L PR[91] R[100]mm/sec CNT100;
   1:  PR[91,1] = PR[90,1] + -9.546;
   1:  PR[91,2] = PR[90,2] + 22.356;
   1:  PR[91,3] = PR[90,3] + 59.256;
   1:L PR[91] R[100]mm/sec CNT100;
   1:  PR[91,1] = PR[90,1] + -10.679;
   1:  PR[91,2] = PR[90,2] + 21.930;
   1:  PR[91,3] = PR[90,3] + 59.267;
   1:L PR[91] R[100]mm/sec CNT100;
   1:  PR[91,1] = PR[90,1] + -11.953;
   1:  PR[91,2] = PR[90,2] + 21.367;
   1:  PR[91,3] = PR[90,3] + 59.277;
   1:L PR[91] R[100]mm/sec CNT100;
   1:  PR[91,1] = PR[90,1] + -12.874;
   1:  PR[91,2] = PR[90,2] + 20.908;
   1:  PR[91,3] = PR[90,3] + 59.289;
   1:L PR[91] R[100]mm/sec CNT100;
   1:  PR[91,1] = PR[90,1] + -13.928;
   1:  PR[91,2] = PR[90,2] + 20.314;
   1:  PR[91,3] = PR[90,3] + 59.298;
   1:L PR[91] R[100]mm/sec CNT100;
   1:  PR[91,1] = PR[90,1] + -14.948;
   1:  PR[91,2] = PR[90,2] + 19.668;
   1:  PR[91,3] = PR[90,3] + 59.308;
   1:L PR[91] R[100]mm/sec CNT100;
   1:  PR[91,1] = PR[90,1] + -15.933;
   1:  PR[91,2] = PR[90,2] + 18.971;
   1:  PR[91,3] = PR[90,3] + 59.319;
   1:L PR[91] R[100]mm/sec CNT100;
   1:  PR[91,1] = PR[90,1] + -16.880;
   1:  PR[91,2] = PR[90,2] + 18.225;
   1:  PR[91,3] = PR[90,3] + 59.329;
   1:L PR[91] R[100]mm/sec CNT100;
   1:  PR[91,1] = PR[90,1] + -17.786;
   1:  PR[91,2] = PR[90,2] + 17.432;
   1:  PR[91,3] = PR[90,3] + 59.340;
   1:L PR[91] R[100]mm/sec CNT100;
   1:  PR[91,1] = PR[90,1] + -18.649;
   1:  PR[91,2] = PR[90,2] + 16.595;
   1:  PR[91,3] = PR[90,3] + 59.350;
   1:L PR[91] R[100]mm/sec CNT100;
   1:  PR[91,1] = PR[90,1] + -19.468;
   1:  PR[91,2] = PR[90,2] + 15.715;
   1:  PR[91,3] = PR[90,3] + 59.361;
   1:L PR[91] R[100]mm/sec CNT100;
   1:  PR[91,1] = PR[90,1] + -20.239;
   1:  PR[91,2] = PR[90,2] + 14.795;
   1:  PR[91,3] = PR[90,3] + 59.371;
   1:L PR[91] R[100]mm/sec CNT100;
   1:  PR[91,1] = PR[90,1] + -20.960;
   1:  PR[91,2] = PR[90,2] + 13.838;
   1:  PR[91,3] = PR[90,3] + 59.382;
   1:L PR[91] R[100]mm/sec CNT100;
   1:  PR[91,1] = PR[90,1] + -21.642;
   1:  PR[91,2] = PR[90,2] + 12.829;
   1:  PR[91,3] = PR[90,3] + 59.392;
   1:L PR[91] R[100]mm/sec CNT100;
   1:  PR[91,1] = PR[90,1] + -22.254;
   1:  PR[91,2] = PR[90,2] + 11.813;
   1:  PR[91,3] = PR[90,3] + 59.402;
   1:L PR[91] R[100]mm/sec CNT100;
   1:  PR[91,1] = PR[90,1] + -22.814;
   1:  PR[91,2] = PR[90,2] + 10.767;
   1:  PR[91,3] = PR[90,3] + 59.413;
   1:L PR[91] R[100]mm/sec CNT100;
   1:  PR[91,1] = PR[90,1] + -23.323;
   1:  PR[91,2] = PR[90,2] + 9.686;
   1:  PR[91,3] = PR[90,3] + 59.423;
   1:L PR[91] R[100]mm/sec CNT100;
   1:  PR[91,1] = PR[90,1] + -23.775;
   1:  PR[91,2] = PR[90,2] + 8.582;
   1:  PR[91,3] = PR[90,3] + 59.433;
   1:L PR[91] R[100]mm/sec CNT100;
   1:  PR[91,1] = PR[90,1] + -24.169;
   1:  PR[91,2] = PR[90,2] + 7.457;
   1:  PR[91,3] = PR[90,3] + 59.444;
   1:L PR[91] R[100]mm/sec CNT100;
   1:  PR[91,1] = PR[90,1] + -24.504;
   1:  PR[91,2] = PR[90,2] + 6.315;
   1:  PR[91,3] = PR[90,3] + 59.454;
   1:L PR[91] R[100]mm/sec CNT100;
   1:  PR[91,1] = PR[90,1] + -24.779;
   1:  PR[91,2] = PR[90,2] + 5.157;
   1:  PR[91,3] = PR[90,3] + 59.464;
   1:L PR[91] R[100]mm/sec CNT100;
   1:  PR[91,1] = PR[90,1] + -24.994;
   1:  PR[91,2] = PR[90,2] + 3.987;
   1:  PR[91,3] = PR[90,3] + 59.475;
   1:L PR[91] R[100]mm/sec CNT100;
   1:  PR[91,1] = PR[90,1] + -25.148;
   1:  PR[91,2] = PR[90,2] + 2.807;
   1:  PR[91,3] = PR[90,3] + 59.485;
   1:L PR[91] R[100]mm/sec CNT100;
   1:  PR[91,1] = PR[90,1] + -25.240;
   1:  PR[91,2] = PR[90,2] + 1.620;
   1:  PR[91,3] = PR[90,3] + 59.495;
   1:L PR[91] R[100]mm/sec CNT100;
   1:  PR[91,1] = PR[90,1] + -25.271;
   1:  PR[91,2] = PR[90,2] + 0.428;
   1:  PR[91,3] = PR[90,3] + 59.506;
   1:L PR[91] R[100]mm/sec CNT100;
   1:  PR[91,1] = PR[90,1] + -25.240;
   1:  PR[91,2] = PR[90,2] + -0.765;
   1:  PR[91,3] = PR[90,3] + 59.516;
   1:L PR[91] R[100]mm/sec CNT100;
   1:  PR[91,1] = PR[90,1] + -25.148;
   1:  PR[91,2] = PR[90,2] + -1.952;
   1:  PR[91,3] = PR[90,3] + 59.526;
   1:L PR[91] R[100]mm/sec CNT100;
   1:  PR[91,1] = PR[90,1] + -24.994;
   1:  PR[91,2] = PR[90,2] + -3.132;
   1:  PR[91,3] = PR[90,3] + 59.537;
   1:L PR[91] R[100]mm/sec CNT100;
   1:  PR[91,1] = PR[90,1] + -24.779;
   1:  PR[91,2] = PR[90,2] + -4.302;
   1:  PR[91,3] = PR[90,3] + 59.547;
   1:L PR[91] R[100]mm/sec CNT100;
   1:  PR[91,1] = PR[90,1] + -24.504;
   1:  PR[91,2] = PR[90,2] + -5.459;
   1:  PR[91,3] = PR[90,3] + 59.557;
   1:L PR[91] R[100]mm/sec CNT100;
   1:  PR[91,1] = PR[90,1] + -24.169;
   1:  PR[91,2] = PR[90,2] + -6.601;
   1:  PR[91,3] = PR[90,3] + 59.568;
   1:L PR[91] R[100]mm/sec CNT100;
   1:  PR[91,1] = PR[90,1] + -23.769;
   1:  PR[91,2] = PR[90,2] + -7.741;
   1:  PR[91,3] = PR[90,3] + 59.578;
   1:L PR[91] R[100]mm/sec CNT100;
   1:  PR[91,1] = PR[90,1] + -23.319;
   1:  PR[91,2] = PR[90,2] + -8.838;
   1:  PR[91,3] = PR[90,3] + 59.588;
   1:L PR[91] R[100]mm/sec CNT100;
   1:  PR[91,1] = PR[90,1] + -22.815;
   1:  PR[91,2] = PR[90,2] + -9.911;
   1:  PR[91,3] = PR[90,3] + 59.599;
   1:L PR[91] R[100]mm/sec CNT100;
   1:  PR[91,1] = PR[90,1] + -22.251;
   1:  PR[91,2] = PR[90,2] + -10.965;
   1:  PR[91,3] = PR[90,3] + 59.609;
   1:L PR[91] R[100]mm/sec CNT100;
   1:  PR[91,1] = PR[90,1] + -21.632;
   1:  PR[91,2] = PR[90,2] + -11.989;
   1:  PR[91,3] = PR[90,3] + 59.619;
   1:L PR[91] R[100]mm/sec CNT100;
   1:  PR[91,1] = PR[90,1] + -20.961;
   1:  PR[91,2] = PR[90,2] + -12.982;
   1:  PR[91,3] = PR[90,3] + 59.630;
   1:L PR[91] R[100]mm/sec CNT100;
   1:  PR[91,1] = PR[90,1] + -20.239;
   1:  PR[91,2] = PR[90,2] + -13.939;
   1:  PR[91,3] = PR[90,3] + 59.640;
   1:L PR[91] R[100]mm/sec CNT100;
   1:  PR[91,1] = PR[90,1] + -19.469;
   1:  PR[91,2] = PR[90,2] + -14.859;
   1:  PR[91,3] = PR[90,3] + 59.650;
   1:L PR[91] R[100]mm/sec CNT100;
   1:  PR[91,1] = PR[90,1] + -18.650;
   1:  PR[91,2] = PR[90,2] + -15.739;
   1:  PR[91,3] = PR[90,3] + 59.661;
   1:L PR[91] R[100]mm/sec CNT100;
   1:  PR[91,1] = PR[90,1] + -17.787;
   1:  PR[91,2] = PR[90,2] + -16.576;
   1:  PR[91,3] = PR[90,3] + 59.671;
   1:L PR[91] R[100]mm/sec CNT100;
   1:  PR[91,1] = PR[90,1] + -16.881;
   1:  PR[91,2] = PR[90,2] + -17.369;
   1:  PR[91,3] = PR[90,3] + 59.682;
   1:L PR[91] R[100]mm/sec CNT100;
   1:  PR[91,1] = PR[90,1] + -15.935;
   1:  PR[91,2] = PR[90,2] + -18.114;
   1:  PR[91,3] = PR[90,3] + 59.692;
   1:L PR[91] R[100]mm/sec CNT100;
   1:  PR[91,1] = PR[90,1] + -14.950;
   1:  PR[91,2] = PR[90,2] + -18.812;
   1:  PR[91,3] = PR[90,3] + 59.703;
   1:L PR[91] R[100]mm/sec CNT100;
   1:  PR[91,1] = PR[90,1] + -13.929;
   1:  PR[91,2] = PR[90,2] + -19.458;
   1:  PR[91,3] = PR[90,3] + 59.713;
   1:L PR[91] R[100]mm/sec CNT100;
   1:  PR[91,1] = PR[90,1] + -13.019;
   1:  PR[91,2] = PR[90,2] + -19.972;
   1:  PR[91,3] = PR[90,3] + 59.724;
   1:L PR[91] R[100]mm/sec CNT100;
   1:  PR[91,1] = PR[90,1] + -11.792;
   1:  PR[91,2] = PR[90,2] + -20.591;
   1:  PR[91,3] = PR[90,3] + 59.733;
   1:L PR[91] R[100]mm/sec CNT100;
   1:  PR[91,1] = PR[90,1] + -10.683;
   1:  PR[91,2] = PR[90,2] + -21.074;
   1:  PR[91,3] = PR[90,3] + 59.745;
   1:L PR[91] R[100]mm/sec CNT100;
   1:  PR[91,1] = PR[90,1] + -9.548;
   1:  PR[91,2] = PR[90,2] + -21.500;
   1:  PR[91,3] = PR[90,3] + 59.755;
   1:L PR[91] R[100]mm/sec CNT100;
   1:  PR[91,1] = PR[90,1] + -8.392;
   1:  PR[91,2] = PR[90,2] + -21.867;
   1:  PR[91,3] = PR[90,3] + 59.766;
   1:L PR[91] R[100]mm/sec CNT100;
   1:  PR[91,1] = PR[90,1] + -7.218;
   1:  PR[91,2] = PR[90,2] + -22.175;
   1:  PR[91,3] = PR[90,3] + 59.776;
   1:L PR[91] R[100]mm/sec CNT100;
   1:  PR[91,1] = PR[90,1] + -6.029;
   1:  PR[91,2] = PR[90,2] + -22.422;
   1:  PR[91,3] = PR[90,3] + 59.787;
   1:L PR[91] R[100]mm/sec CNT100;
   1:  PR[91,1] = PR[90,1] + -4.827;
   1:  PR[91,2] = PR[90,2] + -22.607;
   1:  PR[91,3] = PR[90,3] + 59.797;
   1:L PR[91] R[100]mm/sec CNT100;
   1:  PR[91,1] = PR[90,1] + -3.618;
   1:  PR[91,2] = PR[90,2] + -22.731;
   1:  PR[91,3] = PR[90,3] + 59.808;
   1:L PR[91] R[100]mm/sec CNT100;
   1:  PR[91,1] = PR[90,1] + -2.403;
   1:  PR[91,2] = PR[90,2] + -22.792;
   1:  PR[91,3] = PR[90,3] + 59.818;
   1:L PR[91] R[100]mm/sec CNT100;
   1:  PR[91,1] = PR[90,1] + -1.184;
   1:  PR[91,2] = PR[90,2] + -22.790;
   1:  PR[91,3] = PR[90,3] + 59.829;
   1:L PR[91] R[100]mm/sec CNT100;
   1:  PR[91,1] = PR[90,1] + -0.290;
   1:  PR[91,2] = PR[90,2] + -22.747;
   1:  PR[91,3] = PR[90,3] + 59.839;
   1:L PR[91] R[100]mm/sec CNT100;
   1:  PR[91,1] = PR[90,1] + 0.051;
   1:  PR[91,3] = PR[90,3] + 59.847;
   1:L PR[91] R[100]mm/sec CNT100;
   1:  PR[91] = PR[90];
   1:  PR[91,1] = PR[90,1] + 0.315;
   1:  PR[91,2] = PR[90,2] + -23.100;
   1:  PR[91,3] = PR[90,3] + 61.180;
   1:L PR[91] R[100]mm/sec CNT100;
   1:  PR[91,1] = PR[90,1] + 1.553;
   1:  PR[91,2] = PR[90,2] + -23.110;
   1:  PR[91,3] = PR[90,3] + 59.853;
   1:L PR[91] R[100]mm/sec CNT100;
   1:  PR[91,1] = PR[90,1] + 2.784;
   1:  PR[91,2] = PR[90,2] + -23.055;
   1:  PR[91,3] = PR[90,3] + 59.863;
   1:L PR[91] R[100]mm/sec CNT100;
   1:  PR[91,1] = PR[90,1] + 4.010;
   1:  PR[91,2] = PR[90,2] + -22.937;
   1:  PR[91,3] = PR[90,3] + 59.874;
   1:L PR[91] R[100]mm/sec CNT100;
   1:  PR[91,1] = PR[90,1] + 5.229;
   1:  PR[91,2] = PR[90,2] + -22.755;
   1:  PR[91,3] = PR[90,3] + 59.885;
   1:L PR[91] R[100]mm/sec CNT100;
   1:  PR[91,1] = PR[90,1] + 6.085;
   1:  PR[91,2] = PR[90,2] + -22.585;
   1:  PR[91,3] = PR[90,3] + 59.896;
   1:L PR[91] R[100]mm/sec CNT100;
   1:  PR[91,1] = PR[90,1] + 6.432;
   1:  PR[91,2] = PR[90,2] + -22.512;
   1:  PR[91,3] = PR[90,3] + 59.903;
   1:L PR[91] R[100]mm/sec CNT100;
   1:  PR[91,1] = PR[90,1] + 7.626;
   1:  PR[91,2] = PR[90,2] + -22.206;
   1:  PR[91,3] = PR[90,3] + 59.906;
   1:L PR[91] R[100]mm/sec CNT100;
   1:  PR[91,1] = PR[90,1] + 8.800;
   1:  PR[91,2] = PR[90,2] + -21.839;
   1:  PR[91,3] = PR[90,3] + 59.917;
   1:L PR[91] R[100]mm/sec CNT100;
   1:  PR[91,1] = PR[90,1] + 9.953;
   1:  PR[91,2] = PR[90,2] + -21.412;
   1:  PR[91,3] = PR[90,3] + 59.928;
   1:L PR[91] R[100]mm/sec CNT100;
   1:  PR[91,1] = PR[90,1] + 11.081;
   1:  PR[91,2] = PR[90,2] + -20.927;
   1:  PR[91,3] = PR[90,3] + 59.938;
   1:L PR[91] R[100]mm/sec CNT100;
   1:  PR[91,1] = PR[90,1] + 12.182;
   1:  PR[91,2] = PR[90,2] + -20.385;
   1:  PR[91,3] = PR[90,3] + 59.949;
   1:L PR[91] R[100]mm/sec CNT100;
   1:  PR[91,1] = PR[90,1] + 13.253;
   1:  PR[91,2] = PR[90,2] + -19.787;
   1:  PR[91,3] = PR[90,3] + 59.960;
   1:L PR[91] R[100]mm/sec CNT100;
   1:  PR[91,1] = PR[90,1] + 14.291;
   1:  PR[91,2] = PR[90,2] + -19.134;
   1:  PR[91,3] = PR[90,3] + 59.970;
   1:L PR[91] R[100]mm/sec CNT100;
   1:  PR[91,1] = PR[90,1] + 15.293;
   1:  PR[91,2] = PR[90,2] + -18.430;
   1:  PR[91,3] = PR[90,3] + 59.981;
   1:L PR[91] R[100]mm/sec CNT100;
   1:  PR[91,1] = PR[90,1] + 16.257;
   1:  PR[91,2] = PR[90,2] + -17.676;
   1:  PR[91,3] = PR[90,3] + 59.991;
   1:L PR[91] R[100]mm/sec CNT100;
   1:  PR[91,1] = PR[90,1] + 17.181;
   1:  PR[91,2] = PR[90,2] + -16.873;
   1:  PR[91,3] = PR[90,3] + 60.002;
   1:L PR[91] R[100]mm/sec CNT100;
   1:  PR[91,1] = PR[90,1] + 17.714;
   1:  PR[91,2] = PR[90,2] + -16.359;
   1:  PR[91,3] = PR[90,3] + 60.013;
   1:L PR[91] R[100]mm/sec CNT100;
   1:  PR[91,1] = PR[90,1] + 18.059;
   1:  PR[91,2] = PR[90,2] + -16.025;
   1:  PR[91,3] = PR[90,3] + 60.019;
   1:L PR[91] R[100]mm/sec CNT100;
   1:  PR[91,1] = PR[90,1] + 18.893;
   1:  PR[91,2] = PR[90,2] + -15.132;
   1:  PR[91,3] = PR[90,3] + 60.023;
   1:L PR[91] R[100]mm/sec CNT100;
   1:  PR[91,1] = PR[90,1] + 19.680;
   1:  PR[91,2] = PR[90,2] + -14.198;
   1:  PR[91,3] = PR[90,3] + 60.034;
   1:L PR[91] R[100]mm/sec CNT100;
   1:  PR[91,1] = PR[90,1] + 20.416;
   1:  PR[91,2] = PR[90,2] + -13.226;
   1:  PR[91,3] = PR[90,3] + 60.044;
   1:L PR[91] R[100]mm/sec CNT100;
   1:  PR[91,1] = PR[90,1] + 21.100;
   1:  PR[91,2] = PR[90,2] + -12.218;
   1:  PR[91,3] = PR[90,3] + 60.055;
   1:L PR[91] R[100]mm/sec CNT100;
   1:  PR[91,1] = PR[90,1] + 21.731;
   1:  PR[91,2] = PR[90,2] + -11.176;
   1:  PR[91,3] = PR[90,3] + 60.066;
   1:L PR[91] R[100]mm/sec CNT100;
   1:  PR[91,1] = PR[90,1] + 22.307;
   1:  PR[91,2] = PR[90,2] + -10.104;
   1:  PR[91,3] = PR[90,3] + 60.076;
   1:L PR[91] R[100]mm/sec CNT100;
   1:  PR[91,1] = PR[90,1] + 22.826;
   1:  PR[91,2] = PR[90,2] + -9.005;
   1:  PR[91,3] = PR[90,3] + 60.087;
   1:L PR[91] R[100]mm/sec CNT100;
   1:  PR[91,1] = PR[90,1] + 23.287;
   1:  PR[91,2] = PR[90,2] + -7.881;
   1:  PR[91,3] = PR[90,3] + 60.097;
   1:L PR[91] R[100]mm/sec CNT100;
   1:  PR[91,1] = PR[90,1] + 23.689;
   1:  PR[91,2] = PR[90,2] + -6.735;
   1:  PR[91,3] = PR[90,3] + 60.108;
   1:L PR[91] R[100]mm/sec CNT100;
   1:  PR[91,1] = PR[90,1] + 24.031;
   1:  PR[91,2] = PR[90,2] + -5.571;
   1:  PR[91,3] = PR[90,3] + 60.118;
   1:L PR[91] R[100]mm/sec CNT100;
   1:  PR[91,1] = PR[90,1] + 24.312;
   1:  PR[91,2] = PR[90,2] + -4.391;
   1:  PR[91,3] = PR[90,3] + 60.129;
   1:L PR[91] R[100]mm/sec CNT100;
   1:  PR[91,1] = PR[90,1] + 24.531;
   1:  PR[91,2] = PR[90,2] + -3.199;
   1:  PR[91,3] = PR[90,3] + 60.139;
   1:L PR[91] R[100]mm/sec CNT100;
   1:  PR[91,1] = PR[90,1] + 24.688;
   1:  PR[91,2] = PR[90,2] + -1.996;
   1:  PR[91,3] = PR[90,3] + 60.150;
   1:L PR[91] R[100]mm/sec CNT100;
   1:  PR[91,1] = PR[90,1] + 24.783;
   1:  PR[91,2] = PR[90,2] + -0.787;
   1:  PR[91,3] = PR[90,3] + 60.160;
   1:L PR[91] R[100]mm/sec CNT100;
   1:  PR[91,1] = PR[90,1] + 24.811;
   1:  PR[91,2] = PR[90,2] + 0.428;
   1:  PR[91,3] = PR[90,3] + 60.171;
   1:L PR[91] R[100]mm/sec CNT100;
   1:  PR[91,1] = PR[90,1] + 24.783;
   1:  PR[91,2] = PR[90,2] + 1.642;
   1:  PR[91,3] = PR[90,3] + 60.181;
   1:L PR[91] R[100]mm/sec CNT100;
   1:  PR[91,1] = PR[90,1] + 24.688;
   1:  PR[91,2] = PR[90,2] + 2.851;
   1:  PR[91,3] = PR[90,3] + 60.192;
   1:L PR[91] R[100]mm/sec CNT100;
   1:  PR[91,1] = PR[90,1] + 24.531;
   1:  PR[91,2] = PR[90,2] + 4.054;
   1:  PR[91,3] = PR[90,3] + 60.203;
   1:L PR[91] R[100]mm/sec CNT100;
   1:  PR[91,1] = PR[90,1] + 24.312;
   1:  PR[91,2] = PR[90,2] + 5.247;
   1:  PR[91,3] = PR[90,3] + 60.213;
   1:L PR[91] R[100]mm/sec CNT100;
   1:  PR[91,1] = PR[90,1] + 24.031;
   1:  PR[91,2] = PR[90,2] + 6.427;
   1:  PR[91,3] = PR[90,3] + 60.224;
   1:L PR[91] R[100]mm/sec CNT100;
   1:  PR[91,1] = PR[90,1] + 23.689;
   1:  PR[91,2] = PR[90,2] + 7.591;
   1:  PR[91,3] = PR[90,3] + 60.234;
   1:L PR[91] R[100]mm/sec CNT100;
   1:  PR[91,1] = PR[90,1] + 23.287;
   1:  PR[91,2] = PR[90,2] + 8.736;
   1:  PR[91,3] = PR[90,3] + 60.245;
   1:L PR[91] R[100]mm/sec CNT100;
   1:  PR[91,1] = PR[90,1] + 22.826;
   1:  PR[91,2] = PR[90,2] + 9.860;
   1:  PR[91,3] = PR[90,3] + 60.255;
   1:L PR[91] R[100]mm/sec CNT100;
   1:  PR[91,1] = PR[90,1] + 22.306;
   1:  PR[91,2] = PR[90,2] + 10.960;
   1:  PR[91,3] = PR[90,3] + 60.266;
   1:L PR[91] R[100]mm/sec CNT100;
   1:  PR[91,1] = PR[90,1] + 21.731;
   1:  PR[91,2] = PR[90,2] + 12.032;
   1:  PR[91,3] = PR[90,3] + 60.276;
   1:L PR[91] R[100]mm/sec CNT100;
   1:  PR[91,1] = PR[90,1] + 21.100;
   1:  PR[91,2] = PR[90,2] + 13.073;
   1:  PR[91,3] = PR[90,3] + 60.287;
   1:L PR[91] R[100]mm/sec CNT100;
   1:  PR[91,1] = PR[90,1] + 20.415;
   1:  PR[91,2] = PR[90,2] + 14.082;
   1:  PR[91,3] = PR[90,3] + 60.297;
   1:L PR[91] R[100]mm/sec CNT100;
   1:  PR[91,1] = PR[90,1] + 19.679;
   1:  PR[91,2] = PR[90,2] + 15.054;
   1:  PR[91,3] = PR[90,3] + 60.308;
   1:L PR[91] R[100]mm/sec CNT100;
   1:  PR[91,1] = PR[90,1] + 18.893;
   1:  PR[91,2] = PR[90,2] + 15.988;
   1:  PR[91,3] = PR[90,3] + 60.318;
   1:L PR[91] R[100]mm/sec CNT100;
   1:  PR[91,1] = PR[90,1] + 18.059;
   1:  PR[91,2] = PR[90,2] + 16.880;
   1:  PR[91,3] = PR[90,3] + 60.329;
   1:L PR[91] R[100]mm/sec CNT100;
   1:  PR[91,1] = PR[90,1] + 17.179;
   1:  PR[91,2] = PR[90,2] + 17.729;
   1:  PR[91,3] = PR[90,3] + 60.340;
   1:L PR[91] R[100]mm/sec CNT100;
   1:  PR[91,1] = PR[90,1] + 16.257;
   1:  PR[91,2] = PR[90,2] + 18.531;
   1:  PR[91,3] = PR[90,3] + 60.350;
   1:L PR[91] R[100]mm/sec CNT100;
   1:  PR[91,1] = PR[90,1] + 15.293;
   1:  PR[91,2] = PR[90,2] + 19.286;
   1:  PR[91,3] = PR[90,3] + 60.361;
   1:L PR[91] R[100]mm/sec CNT100;
   1:  PR[91,1] = PR[90,1] + 14.290;
   1:  PR[91,2] = PR[90,2] + 19.990;
   1:  PR[91,3] = PR[90,3] + 60.372;
   1:L PR[91] R[100]mm/sec CNT100;
   1:  PR[91,1] = PR[90,1] + 13.252;
   1:  PR[91,2] = PR[90,2] + 20.642;
   1:  PR[91,3] = PR[90,3] + 60.382;
   1:L PR[91] R[100]mm/sec CNT100;
   1:  PR[91,1] = PR[90,1] + 12.181;
   1:  PR[91,2] = PR[90,2] + 21.240;
   1:  PR[91,3] = PR[90,3] + 60.393;
   1:L PR[91] R[100]mm/sec CNT100;
   1:  PR[91,1] = PR[90,1] + 11.078;
   1:  PR[91,2] = PR[90,2] + 21.784;
   1:  PR[91,3] = PR[90,3] + 60.403;
   1:L PR[91] R[100]mm/sec CNT100;
   1:  PR[91,1] = PR[90,1] + 10.709;
   1:  PR[91,2] = PR[90,2] + 21.945;
   1:  PR[91,3] = PR[90,3] + 60.414;
   1:L PR[91] R[100]mm/sec CNT100;
   1:  PR[91,1] = PR[90,1] + 9.952;
   1:  PR[91,2] = PR[90,2] + 22.268;
   1:  PR[91,3] = PR[90,3] + 60.418;
   1:L PR[91] R[100]mm/sec CNT100;
   1:  PR[91,1] = PR[90,1] + 8.799;
   1:  PR[91,2] = PR[90,2] + 22.695;
   1:  PR[91,3] = PR[90,3] + 60.425;
   1:L PR[91] R[100]mm/sec CNT100;
   1:  PR[91,1] = PR[90,1] + 7.625;
   1:  PR[91,2] = PR[90,2] + 23.061;
   1:  PR[91,3] = PR[90,3] + 60.435;
   1:L PR[91] R[100]mm/sec CNT100;
   1:  PR[91,1] = PR[90,1] + 6.433;
   1:  PR[91,2] = PR[90,2] + 23.367;
   1:  PR[91,3] = PR[90,3] + 60.446;
   1:L PR[91] R[100]mm/sec CNT100;
   1:  PR[91,1] = PR[90,1] + 5.227;
   1:  PR[91,2] = PR[90,2] + 23.611;
   1:  PR[91,3] = PR[90,3] + 60.457;
   1:L PR[91] R[100]mm/sec CNT100;
   1:  PR[91,1] = PR[90,1] + 4.009;
   1:  PR[91,2] = PR[90,2] + 23.792;
   1:  PR[91,3] = PR[90,3] + 60.467;
   1:L PR[91] R[100]mm/sec CNT100;
   1:  PR[91,1] = PR[90,1] + 2.782;
   1:  PR[91,2] = PR[90,2] + 23.910;
   1:  PR[91,3] = PR[90,3] + 60.478;
   1:L PR[91] R[100]mm/sec CNT100;
   1:  PR[91,1] = PR[90,1] + 1.553;
   1:  PR[91,2] = PR[90,2] + 23.965;
   1:  PR[91,3] = PR[90,3] + 60.489;
   1:L PR[91] R[100]mm/sec CNT100;
   1:  PR[91,1] = PR[90,1] + -0.240;
   1:  PR[91,2] = PR[90,2] + 23.940;
   1:  PR[91,3] = PR[90,3] + 60.499;
   1:L PR[91] R[100]mm/sec CNT100;
   1:  PR[91,1] = PR[90,1] + -0.553;
   1:  PR[91,2] = PR[90,2] + 23.955;
   1:  PR[91,3] = PR[90,3] + 60.515;
   1:L PR[91] R[100]mm/sec CNT100;
   1:  PR[91,1] = PR[90,1] + -1.790;
   1:  PR[91,2] = PR[90,2] + 23.965;
   1:  PR[91,3] = PR[90,3] + 60.518;
   1:L PR[91] R[100]mm/sec CNT100;
   1:  PR[91,1] = PR[90,1] + -3.021;
   1:  PR[91,2] = PR[90,2] + 23.910;
   1:  PR[91,3] = PR[90,3] + 60.528;
   1:L PR[91] R[100]mm/sec CNT100;
   1:  PR[91,1] = PR[90,1] + -4.247;
   1:  PR[91,2] = PR[90,2] + 23.792;
   1:  PR[91,3] = PR[90,3] + 60.539;
   1:L PR[91] R[100]mm/sec CNT100;
   1:  PR[91,1] = PR[90,1] + -5.465;
   1:  PR[91,2] = PR[90,2] + 23.611;
   1:  PR[91,3] = PR[90,3] + 60.550;
   1:L PR[91] R[100]mm/sec CNT100;
   1:  PR[91,1] = PR[90,1] + -6.672;
   1:  PR[91,2] = PR[90,2] + 23.367;
   1:  PR[91,3] = PR[90,3] + 60.561;
   1:L PR[91] R[100]mm/sec CNT100;
   1:  PR[91,1] = PR[90,1] + -7.864;
   1:  PR[91,2] = PR[90,2] + 23.061;
   1:  PR[91,3] = PR[90,3] + 60.571;
   1:L PR[91] R[100]mm/sec CNT100;
   1:  PR[91,1] = PR[90,1] + -9.038;
   1:  PR[91,2] = PR[90,2] + 22.695;
   1:  PR[91,3] = PR[90,3] + 60.582;
   1:L PR[91] R[100]mm/sec CNT100;
   1:  PR[91,1] = PR[90,1] + -10.190;
   1:  PR[91,2] = PR[90,2] + 22.268;
   1:  PR[91,3] = PR[90,3] + 60.593;
   1:L PR[91] R[100]mm/sec CNT100;
   1:  PR[91,1] = PR[90,1] + -11.319;
   1:  PR[91,2] = PR[90,2] + 21.783;
   1:  PR[91,3] = PR[90,3] + 60.603;
   1:L PR[91] R[100]mm/sec CNT100;
   1:  PR[91,1] = PR[90,1] + -12.420;
   1:  PR[91,2] = PR[90,2] + 21.240;
   1:  PR[91,3] = PR[90,3] + 60.614;
   1:L PR[91] R[100]mm/sec CNT100;
   1:  PR[91,1] = PR[90,1] + -13.491;
   1:  PR[91,2] = PR[90,2] + 20.642;
   1:  PR[91,3] = PR[90,3] + 60.624;
   1:L PR[91] R[100]mm/sec CNT100;
   1:  PR[91,1] = PR[90,1] + -14.529;
   1:  PR[91,2] = PR[90,2] + 19.990;
   1:  PR[91,3] = PR[90,3] + 60.635;
   1:L PR[91] R[100]mm/sec CNT100;
   1:  PR[91,1] = PR[90,1] + -15.531;
   1:  PR[91,2] = PR[90,2] + 19.286;
   1:  PR[91,3] = PR[90,3] + 60.646;
   1:L PR[91] R[100]mm/sec CNT100;
   1:  PR[91,1] = PR[90,1] + -16.496;
   1:  PR[91,2] = PR[90,2] + 18.531;
   1:  PR[91,3] = PR[90,3] + 60.656;
   1:L PR[91] R[100]mm/sec CNT100;
   1:  PR[91,1] = PR[90,1] + -17.063;
   1:  PR[91,2] = PR[90,2] + 18.040;
   1:  PR[91,3] = PR[90,3] + 60.667;
   1:L PR[91] R[100]mm/sec CNT100;
   1:  PR[91,1] = PR[90,1] + -17.417;
   1:  PR[91,2] = PR[90,2] + 17.729;
   1:  PR[91,3] = PR[90,3] + 60.674;
   1:L PR[91] R[100]mm/sec CNT100;
   1:  PR[91,1] = PR[90,1] + -18.298;
   1:  PR[91,2] = PR[90,2] + 16.880;
   1:  PR[91,3] = PR[90,3] + 60.678;
   1:L PR[91] R[100]mm/sec CNT100;
   1:  PR[91,1] = PR[90,1] + -19.131;
   1:  PR[91,2] = PR[90,2] + 15.988;
   1:  PR[91,3] = PR[90,3] + 60.688;
   1:L PR[91] R[100]mm/sec CNT100;
   1:  PR[91,1] = PR[90,1] + -19.918;
   1:  PR[91,2] = PR[90,2] + 15.054;
   1:  PR[91,3] = PR[90,3] + 60.699;
   1:L PR[91] R[100]mm/sec CNT100;
   1:  PR[91,1] = PR[90,1] + -20.654;
   1:  PR[91,2] = PR[90,2] + 14.082;
   1:  PR[91,3] = PR[90,3] + 60.709;
   1:L PR[91] R[100]mm/sec CNT100;
   1:  PR[91,1] = PR[90,1] + -21.338;
   1:  PR[91,2] = PR[90,2] + 13.074;
   1:  PR[91,3] = PR[90,3] + 60.720;
   1:L PR[91] R[100]mm/sec CNT100;
   1:  PR[91,1] = PR[90,1] + -21.969;
   1:  PR[91,2] = PR[90,2] + 12.032;
   1:  PR[91,3] = PR[90,3] + 60.731;
   1:L PR[91] R[100]mm/sec CNT100;
   1:  PR[91,1] = PR[90,1] + -22.545;
   1:  PR[91,2] = PR[90,2] + 10.960;
   1:  PR[91,3] = PR[90,3] + 60.741;
   1:L PR[91] R[100]mm/sec CNT100;
   1:  PR[91,1] = PR[90,1] + -23.064;
   1:  PR[91,2] = PR[90,2] + 9.860;
   1:  PR[91,3] = PR[90,3] + 60.752;
   1:L PR[91] R[100]mm/sec CNT100;
   1:  PR[91,1] = PR[90,1] + -23.525;
   1:  PR[91,2] = PR[90,2] + 8.736;
   1:  PR[91,3] = PR[90,3] + 60.762;
   1:L PR[91] R[100]mm/sec CNT100;
   1:  PR[91,1] = PR[90,1] + -23.928;
   1:  PR[91,2] = PR[90,2] + 7.590;
   1:  PR[91,3] = PR[90,3] + 60.773;
   1:L PR[91] R[100]mm/sec CNT100;
   1:  PR[91,1] = PR[90,1] + -24.270;
   1:  PR[91,2] = PR[90,2] + 6.426;
   1:  PR[91,3] = PR[90,3] + 60.783;
   1:L PR[91] R[100]mm/sec CNT100;
   1:  PR[91,1] = PR[90,1] + -24.551;
   1:  PR[91,2] = PR[90,2] + 5.246;
   1:  PR[91,3] = PR[90,3] + 60.794;
   1:L PR[91] R[100]mm/sec CNT100;
   1:  PR[91,1] = PR[90,1] + -24.770;
   1:  PR[91,2] = PR[90,2] + 4.054;
   1:  PR[91,3] = PR[90,3] + 60.804;
   1:L PR[91] R[100]mm/sec CNT100;
   1:  PR[91,1] = PR[90,1] + -24.927;
   1:  PR[91,2] = PR[90,2] + 2.851;
   1:  PR[91,3] = PR[90,3] + 60.815;
   1:L PR[91] R[100]mm/sec CNT100;
   1:  PR[91,1] = PR[90,1] + -25.021;
   1:  PR[91,2] = PR[90,2] + 1.642;
   1:  PR[91,3] = PR[90,3] + 60.825;
   1:L PR[91] R[100]mm/sec CNT100;
   1:  PR[91,1] = PR[90,1] + -25.049;
   1:  PR[91,2] = PR[90,2] + 0.428;
   1:  PR[91,3] = PR[90,3] + 60.836;
   1:L PR[91] R[100]mm/sec CNT100;
   1:  PR[91,1] = PR[90,1] + -25.021;
   1:  PR[91,2] = PR[90,2] + -0.787;
   1:  PR[91,3] = PR[90,3] + 60.846;
   1:L PR[91] R[100]mm/sec CNT100;
   1:  PR[91,1] = PR[90,1] + -24.927;
   1:  PR[91,2] = PR[90,2] + -1.996;
   1:  PR[91,3] = PR[90,3] + 60.857;
   1:L PR[91] R[100]mm/sec CNT100;
   1:  PR[91,1] = PR[90,1] + -24.770;
   1:  PR[91,2] = PR[90,2] + -3.198;
   1:  PR[91,3] = PR[90,3] + 60.868;
   1:L PR[91] R[100]mm/sec CNT100;
   1:  PR[91,1] = PR[90,1] + -24.551;
   1:  PR[91,2] = PR[90,2] + -4.391;
   1:  PR[91,3] = PR[90,3] + 60.878;
   1:L PR[91] R[100]mm/sec CNT100;
   1:  PR[91,1] = PR[90,1] + -24.270;
   1:  PR[91,2] = PR[90,2] + -5.571;
   1:  PR[91,3] = PR[90,3] + 60.889;
   1:L PR[91] R[100]mm/sec CNT100;
   1:  PR[91,1] = PR[90,1] + -23.928;
   1:  PR[91,2] = PR[90,2] + -6.735;
   1:  PR[91,3] = PR[90,3] + 60.899;
   1:L PR[91] R[100]mm/sec CNT100;
   1:  PR[91,1] = PR[90,1] + -23.526;
   1:  PR[91,2] = PR[90,2] + -7.880;
   1:  PR[91,3] = PR[90,3] + 60.910;
   1:L PR[91] R[100]mm/sec CNT100;
   1:  PR[91,1] = PR[90,1] + -23.064;
   1:  PR[91,2] = PR[90,2] + -9.005;
   1:  PR[91,3] = PR[90,3] + 60.920;
   1:L PR[91] R[100]mm/sec CNT100;
   1:  PR[91,1] = PR[90,1] + -22.545;
   1:  PR[91,2] = PR[90,2] + -10.104;
   1:  PR[91,3] = PR[90,3] + 60.931;
   1:L PR[91] R[100]mm/sec CNT100;
   1:  PR[91,1] = PR[90,1] + -21.969;
   1:  PR[91,2] = PR[90,2] + -11.177;
   1:  PR[91,3] = PR[90,3] + 60.941;
   1:L PR[91] R[100]mm/sec CNT100;
   1:  PR[91,1] = PR[90,1] + -21.339;
   1:  PR[91,2] = PR[90,2] + -12.218;
   1:  PR[91,3] = PR[90,3] + 60.952;
   1:L PR[91] R[100]mm/sec CNT100;
   1:  PR[91,1] = PR[90,1] + -20.654;
   1:  PR[91,2] = PR[90,2] + -13.226;
   1:  PR[91,3] = PR[90,3] + 60.962;
   1:L PR[91] R[100]mm/sec CNT100;
   1:  PR[91,1] = PR[90,1] + -19.918;
   1:  PR[91,2] = PR[90,2] + -14.199;
   1:  PR[91,3] = PR[90,3] + 60.973;
   1:L PR[91] R[100]mm/sec CNT100;
   1:  PR[91,1] = PR[90,1] + -19.132;
   1:  PR[91,2] = PR[90,2] + -15.132;
   1:  PR[91,3] = PR[90,3] + 60.983;
   1:L PR[91] R[100]mm/sec CNT100;
   1:  PR[91,1] = PR[90,1] + -18.298;
   1:  PR[91,2] = PR[90,2] + -16.024;
   1:  PR[91,3] = PR[90,3] + 60.994;
   1:L PR[91] R[100]mm/sec CNT100;
   1:  PR[91,1] = PR[90,1] + -17.419;
   1:  PR[91,2] = PR[90,2] + -16.873;
   1:  PR[91,3] = PR[90,3] + 61.005;
   1:L PR[91] R[100]mm/sec CNT100;
   1:  PR[91,1] = PR[90,1] + -16.496;
   1:  PR[91,2] = PR[90,2] + -17.676;
   1:  PR[91,3] = PR[90,3] + 61.015;
   1:L PR[91] R[100]mm/sec CNT100;
   1:  PR[91,1] = PR[90,1] + -15.532;
   1:  PR[91,2] = PR[90,2] + -18.430;
   1:  PR[91,3] = PR[90,3] + 61.026;
   1:L PR[91] R[100]mm/sec CNT100;
   1:  PR[91,1] = PR[90,1] + -14.530;
   1:  PR[91,2] = PR[90,2] + -19.134;
   1:  PR[91,3] = PR[90,3] + 61.037;
   1:L PR[91] R[100]mm/sec CNT100;
   1:  PR[91,1] = PR[90,1] + -13.492;
   1:  PR[91,2] = PR[90,2] + -19.787;
   1:  PR[91,3] = PR[90,3] + 61.047;
   1:L PR[91] R[100]mm/sec CNT100;
   1:  PR[91,1] = PR[90,1] + -12.421;
   1:  PR[91,2] = PR[90,2] + -20.385;
   1:  PR[91,3] = PR[90,3] + 61.058;
   1:L PR[91] R[100]mm/sec CNT100;
   1:  PR[91,1] = PR[90,1] + -11.319;
   1:  PR[91,2] = PR[90,2] + -20.927;
   1:  PR[91,3] = PR[90,3] + 61.068;
   1:L PR[91] R[100]mm/sec CNT100;
   1:  PR[91,1] = PR[90,1] + -10.189;
   1:  PR[91,2] = PR[90,2] + -21.413;
   1:  PR[91,3] = PR[90,3] + 61.079;
   1:L PR[91] R[100]mm/sec CNT100;
   1:  PR[91,1] = PR[90,1] + -9.824;
   1:  PR[91,2] = PR[90,2] + -21.551;
   1:  PR[91,3] = PR[90,3] + 61.090;
   1:L PR[91] R[100]mm/sec CNT100;
   1:  PR[91,1] = PR[90,1] + -9.039;
   1:  PR[91,2] = PR[90,2] + -21.839;
   1:  PR[91,3] = PR[90,3] + 61.093;
   1:L PR[91] R[100]mm/sec CNT100;
   1:  PR[91,1] = PR[90,1] + -7.865;
   1:  PR[91,2] = PR[90,2] + -22.206;
   1:  PR[91,3] = PR[90,3] + 61.100;
   1:L PR[91] R[100]mm/sec CNT100;
   1:  PR[91,1] = PR[90,1] + -6.673;
   1:  PR[91,2] = PR[90,2] + -22.512;
   1:  PR[91,3] = PR[90,3] + 61.111;
   1:L PR[91] R[100]mm/sec CNT100;
   1:  PR[91,1] = PR[90,1] + -5.466;
   1:  PR[91,2] = PR[90,2] + -22.756;
   1:  PR[91,3] = PR[90,3] + 61.122;
   1:L PR[91] R[100]mm/sec CNT100;
   1:  PR[91,1] = PR[90,1] + -4.248;
   1:  PR[91,2] = PR[90,2] + -22.937;
   1:  PR[91,3] = PR[90,3] + 61.132;
   1:L PR[91] R[100]mm/sec CNT100;
   1:  PR[91,1] = PR[90,1] + -3.022;
   1:  PR[91,2] = PR[90,2] + -23.055;
   1:  PR[91,3] = PR[90,3] + 61.143;
   1:L PR[91] R[100]mm/sec CNT100;
   1:  PR[91,1] = PR[90,1] + -1.793;
   1:  PR[91,2] = PR[90,2] + -23.110;
   1:  PR[91,3] = PR[90,3] + 61.154;
   1:L PR[91] R[100]mm/sec CNT100;
   1:  PR[91,1] = PR[90,1] + 0.001;
   1:  PR[91,2] = PR[90,2] + -23.085;
   1:  PR[91,3] = PR[90,3] + 61.164;
   1:L PR[91] R[100]mm/sec CNT100;
   1:  PR[91] = PR[90];
   1:  PR[91,1] = PR[90,1] + 2.196;
   1:  PR[91,2] = PR[90,2] + -23.385;
   1:  PR[91,3] = PR[90,3] + 62.510;
   1:L PR[91] R[100]mm/sec CNT100;
   1:  PR[91,1] = PR[90,1] + 3.607;
   1:  PR[91,2] = PR[90,2] + -23.251;
   1:  PR[91,3] = PR[90,3] + 61.191;
   1:L PR[91] R[100]mm/sec CNT100;
   1:  PR[91,1] = PR[90,1] + 4.719;
   1:  PR[91,2] = PR[90,2] + -23.087;
   1:  PR[91,3] = PR[90,3] + 61.203;
   1:L PR[91] R[100]mm/sec CNT100;
   1:  PR[91,1] = PR[90,1] + 5.962;
   1:  PR[91,2] = PR[90,2] + -22.839;
   1:  PR[91,3] = PR[90,3] + 61.213;
   1:L PR[91] R[100]mm/sec CNT100;
   1:  PR[91,1] = PR[90,1] + 7.190;
   1:  PR[91,2] = PR[90,2] + -22.526;
   1:  PR[91,3] = PR[90,3] + 61.224;
   1:L PR[91] R[100]mm/sec CNT100;
   1:  PR[91,1] = PR[90,1] + 8.276;
   1:  PR[91,2] = PR[90,2] + -22.190;
   1:  PR[91,3] = PR[90,3] + 61.235;
   1:L PR[91] R[100]mm/sec CNT100;
   1:  PR[91,1] = PR[90,1] + 9.467;
   1:  PR[91,2] = PR[90,2] + -21.755;
   1:  PR[91,3] = PR[90,3] + 61.245;
   1:L PR[91] R[100]mm/sec CNT100;
   1:  PR[91,1] = PR[90,1] + 10.630;
   1:  PR[91,2] = PR[90,2] + -21.260;
   1:  PR[91,3] = PR[90,3] + 61.256;
   1:L PR[91] R[100]mm/sec CNT100;
   1:  PR[91,1] = PR[90,1] + 11.764;
   1:  PR[91,2] = PR[90,2] + -20.705;
   1:  PR[91,3] = PR[90,3] + 61.267;
   1:L PR[91] R[100]mm/sec CNT100;
   1:  PR[91,1] = PR[90,1] + 12.866;
   1:  PR[91,2] = PR[90,2] + -20.092;
   1:  PR[91,3] = PR[90,3] + 61.278;
   1:L PR[91] R[100]mm/sec CNT100;
   1:  PR[91,1] = PR[90,1] + 13.933;
   1:  PR[91,2] = PR[90,2] + -19.422;
   1:  PR[91,3] = PR[90,3] + 61.289;
   1:L PR[91] R[100]mm/sec CNT100;
   1:  PR[91,1] = PR[90,1] + 14.880;
   1:  PR[91,2] = PR[90,2] + -18.760;
   1:  PR[91,3] = PR[90,3] + 61.300;
   1:L PR[91] R[100]mm/sec CNT100;
   1:  PR[91,1] = PR[90,1] + 15.875;
   1:  PR[91,2] = PR[90,2] + -17.986;
   1:  PR[91,3] = PR[90,3] + 61.310;
   1:L PR[91] R[100]mm/sec CNT100;
   1:  PR[91,1] = PR[90,1] + 16.826;
   1:  PR[91,2] = PR[90,2] + -17.163;
   1:  PR[91,3] = PR[90,3] + 61.321;
   1:L PR[91] R[100]mm/sec CNT100;
   1:  PR[91,1] = PR[90,1] + 17.736;
   1:  PR[91,2] = PR[90,2] + -16.287;
   1:  PR[91,3] = PR[90,3] + 61.332;
   1:L PR[91] R[100]mm/sec CNT100;
   1:  PR[91,1] = PR[90,1] + 18.538;
   1:  PR[91,2] = PR[90,2] + -15.433;
   1:  PR[91,3] = PR[90,3] + 61.343;
   1:L PR[91] R[100]mm/sec CNT100;
   1:  PR[91,1] = PR[90,1] + 19.408;
   1:  PR[91,2] = PR[90,2] + -14.401;
   1:  PR[91,3] = PR[90,3] + 61.353;
   1:L PR[91] R[100]mm/sec CNT100;
   1:  PR[91,1] = PR[90,1] + 20.117;
   1:  PR[91,2] = PR[90,2] + -13.466;
   1:  PR[91,3] = PR[90,3] + 61.365;
   1:L PR[91] R[100]mm/sec CNT100;
   1:  PR[91,1] = PR[90,1] + 20.825;
   1:  PR[91,2] = PR[90,2] + -12.425;
   1:  PR[91,3] = PR[90,3] + 61.375;
   1:L PR[91] R[100]mm/sec CNT100;
   1:  PR[91,1] = PR[90,1] + 21.438;
   1:  PR[91,2] = PR[90,2] + -11.417;
   1:  PR[91,3] = PR[90,3] + 61.386;
   1:L PR[91] R[100]mm/sec CNT100;
   1:  PR[91,1] = PR[90,1] + 22.035;
   1:  PR[91,2] = PR[90,2] + -10.310;
   1:  PR[91,3] = PR[90,3] + 61.396;
   1:L PR[91] R[100]mm/sec CNT100;
   1:  PR[91,1] = PR[90,1] + 22.572;
   1:  PR[91,2] = PR[90,2] + -9.176;
   1:  PR[91,3] = PR[90,3] + 61.407;
   1:L PR[91] R[100]mm/sec CNT100;
   1:  PR[91,1] = PR[90,1] + 23.049;
   1:  PR[91,2] = PR[90,2] + -8.017;
   1:  PR[91,3] = PR[90,3] + 61.418;
   1:L PR[91] R[100]mm/sec CNT100;
   1:  PR[91,1] = PR[90,1] + 23.462;
   1:  PR[91,2] = PR[90,2] + -6.835;
   1:  PR[91,3] = PR[90,3] + 61.429;
   1:L PR[91] R[100]mm/sec CNT100;
   1:  PR[91,1] = PR[90,1] + 23.813;
   1:  PR[91,2] = PR[90,2] + -5.634;
   1:  PR[91,3] = PR[90,3] + 61.439;
   1:L PR[91] R[100]mm/sec CNT100;
   1:  PR[91,1] = PR[90,1] + 24.088;
   1:  PR[91,2] = PR[90,2] + -4.479;
   1:  PR[91,3] = PR[90,3] + 61.450;
   1:L PR[91] R[100]mm/sec CNT100;
   1:  PR[91,1] = PR[90,1] + 24.314;
   1:  PR[91,2] = PR[90,2] + -3.249;
   1:  PR[91,3] = PR[90,3] + 61.461;
   1:L PR[91] R[100]mm/sec CNT100;
   1:  PR[91,1] = PR[90,1] + 24.475;
   1:  PR[91,2] = PR[90,2] + -2.009;
   1:  PR[91,3] = PR[90,3] + 61.471;
   1:L PR[91] R[100]mm/sec CNT100;
   1:  PR[91,1] = PR[90,1] + 24.570;
   1:  PR[91,2] = PR[90,2] + -0.762;
   1:  PR[91,3] = PR[90,3] + 61.482;
   1:L PR[91] R[100]mm/sec CNT100;
   1:  PR[91,1] = PR[90,1] + 24.600;
   1:  PR[91,2] = PR[90,2] + 0.427;
   1:  PR[91,3] = PR[90,3] + 61.493;
   1:L PR[91] R[100]mm/sec CNT100;
   1:  PR[91,1] = PR[90,1] + 24.567;
   1:  PR[91,2] = PR[90,2] + 1.678;
   1:  PR[91,3] = PR[90,3] + 61.503;
   1:L PR[91] R[100]mm/sec CNT100;
   1:  PR[91,1] = PR[90,1] + 24.468;
   1:  PR[91,2] = PR[90,2] + 2.925;
   1:  PR[91,3] = PR[90,3] + 61.514;
   1:L PR[91] R[100]mm/sec CNT100;
   1:  PR[91,1] = PR[90,1] + 24.304;
   1:  PR[91,2] = PR[90,2] + 4.166;
   1:  PR[91,3] = PR[90,3] + 61.525;
   1:L PR[91] R[100]mm/sec CNT100;
   1:  PR[91,1] = PR[90,1] + 24.088;
   1:  PR[91,2] = PR[90,2] + 5.334;
   1:  PR[91,3] = PR[90,3] + 61.536;
   1:L PR[91] R[100]mm/sec CNT100;
   1:  PR[91,1] = PR[90,1] + 23.813;
   1:  PR[91,2] = PR[90,2] + 6.488;
   1:  PR[91,3] = PR[90,3] + 61.546;
   1:L PR[91] R[100]mm/sec CNT100;
   1:  PR[91,1] = PR[90,1] + 23.442;
   1:  PR[91,2] = PR[90,2] + 7.754;
   1:  PR[91,3] = PR[90,3] + 61.557;
   1:L PR[91] R[100]mm/sec CNT100;
   1:  PR[91,1] = PR[90,1] + 23.049;
   1:  PR[91,2] = PR[90,2] + 8.871;
   1:  PR[91,3] = PR[90,3] + 61.568;
   1:L PR[91] R[100]mm/sec CNT100;
   1:  PR[91,1] = PR[90,1] + 22.572;
   1:  PR[91,2] = PR[90,2] + 10.031;
   1:  PR[91,3] = PR[90,3] + 61.578;
   1:L PR[91] R[100]mm/sec CNT100;
   1:  PR[91,1] = PR[90,1] + 22.035;
   1:  PR[91,2] = PR[90,2] + 11.166;
   1:  PR[91,3] = PR[90,3] + 61.589;
   1:L PR[91] R[100]mm/sec CNT100;
   1:  PR[91,1] = PR[90,1] + 21.437;
   1:  PR[91,2] = PR[90,2] + 12.272;
   1:  PR[91,3] = PR[90,3] + 61.600;
   1:L PR[91] R[100]mm/sec CNT100;
   1:  PR[91,1] = PR[90,1] + 20.825;
   1:  PR[91,2] = PR[90,2] + 13.280;
   1:  PR[91,3] = PR[90,3] + 61.611;
   1:L PR[91] R[100]mm/sec CNT100;
   1:  PR[91,1] = PR[90,1] + 20.117;
   1:  PR[91,2] = PR[90,2] + 14.321;
   1:  PR[91,3] = PR[90,3] + 61.621;
   1:L PR[91] R[100]mm/sec CNT100;
   1:  PR[91,1] = PR[90,1] + 19.354;
   1:  PR[91,2] = PR[90,2] + 15.324;
   1:  PR[91,3] = PR[90,3] + 61.632;
   1:L PR[91] R[100]mm/sec CNT100;
   1:  PR[91,1] = PR[90,1] + 18.598;
   1:  PR[91,2] = PR[90,2] + 16.221;
   1:  PR[91,3] = PR[90,3] + 61.643;
   1:L PR[91] R[100]mm/sec CNT100;
   1:  PR[91,1] = PR[90,1] + 17.736;
   1:  PR[91,2] = PR[90,2] + 17.143;
   1:  PR[91,3] = PR[90,3] + 61.653;
   1:L PR[91] R[100]mm/sec CNT100;
   1:  PR[91,1] = PR[90,1] + 16.826;
   1:  PR[91,2] = PR[90,2] + 18.019;
   1:  PR[91,3] = PR[90,3] + 61.664;
   1:L PR[91] R[100]mm/sec CNT100;
   1:  PR[91,1] = PR[90,1] + 15.875;
   1:  PR[91,2] = PR[90,2] + 18.841;
   1:  PR[91,3] = PR[90,3] + 61.675;
   1:L PR[91] R[100]mm/sec CNT100;
   1:  PR[91,1] = PR[90,1] + 14.880;
   1:  PR[91,2] = PR[90,2] + 19.615;
   1:  PR[91,3] = PR[90,3] + 61.686;
   1:L PR[91] R[100]mm/sec CNT100;
   1:  PR[91,1] = PR[90,1] + 13.933;
   1:  PR[91,2] = PR[90,2] + 20.278;
   1:  PR[91,3] = PR[90,3] + 61.697;
   1:L PR[91] R[100]mm/sec CNT100;
   1:  PR[91,1] = PR[90,1] + 12.866;
   1:  PR[91,2] = PR[90,2] + 20.947;
   1:  PR[91,3] = PR[90,3] + 61.707;
   1:L PR[91] R[100]mm/sec CNT100;
   1:  PR[91,1] = PR[90,1] + 11.764;
   1:  PR[91,2] = PR[90,2] + 21.560;
   1:  PR[91,3] = PR[90,3] + 61.718;
   1:L PR[91] R[100]mm/sec CNT100;
   1:  PR[91,1] = PR[90,1] + 10.630;
   1:  PR[91,2] = PR[90,2] + 22.115;
   1:  PR[91,3] = PR[90,3] + 61.729;
   1:L PR[91] R[100]mm/sec CNT100;
   1:  PR[91,1] = PR[90,1] + 9.466;
   1:  PR[91,2] = PR[90,2] + 22.611;
   1:  PR[91,3] = PR[90,3] + 61.740;
   1:L PR[91] R[100]mm/sec CNT100;
   1:  PR[91,1] = PR[90,1] + 8.396;
   1:  PR[91,2] = PR[90,2] + 23.004;
   1:  PR[91,3] = PR[90,3] + 61.751;
   1:L PR[91] R[100]mm/sec CNT100;
   1:  PR[91,1] = PR[90,1] + 7.189;
   1:  PR[91,2] = PR[90,2] + 23.381;
   1:  PR[91,3] = PR[90,3] + 61.761;
   1:L PR[91] R[100]mm/sec CNT100;
   1:  PR[91,1] = PR[90,1] + 5.962;
   1:  PR[91,2] = PR[90,2] + 23.694;
   1:  PR[91,3] = PR[90,3] + 61.772;
   1:L PR[91] R[100]mm/sec CNT100;
   1:  PR[91,1] = PR[90,1] + 4.719;
   1:  PR[91,2] = PR[90,2] + 23.942;
   1:  PR[91,3] = PR[90,3] + 61.783;
   1:L PR[91] R[100]mm/sec CNT100;
   1:  PR[91,1] = PR[90,1] + 3.463;
   1:  PR[91,2] = PR[90,2] + 24.125;
   1:  PR[91,3] = PR[90,3] + 61.794;
   1:L PR[91] R[100]mm/sec CNT100;
   1:  PR[91,1] = PR[90,1] + 2.196;
   1:  PR[91,2] = PR[90,2] + 24.240;
   1:  PR[91,3] = PR[90,3] + 61.805;
   1:L PR[91] R[100]mm/sec CNT100;
   1:  PR[91,1] = PR[90,1] + 1.075;
   1:  PR[91,2] = PR[90,2] + 24.287;
   1:  PR[91,3] = PR[90,3] + 61.816;
   1:L PR[91] R[100]mm/sec CNT100;
   1:  PR[91,1] = PR[90,1] + -1.160;
   1:  PR[91,2] = PR[90,2] + 24.289;
   1:  PR[91,3] = PR[90,3] + 61.826;
   1:L PR[91] R[100]mm/sec CNT100;
   1:  PR[91,1] = PR[90,1] + -2.435;
   1:  PR[91,2] = PR[90,2] + 24.240;
   1:  PR[91,3] = PR[90,3] + 61.845;
   1:L PR[91] R[100]mm/sec CNT100;
   1:  PR[91,1] = PR[90,1] + -3.845;
   1:  PR[91,2] = PR[90,2] + 24.106;
   1:  PR[91,3] = PR[90,3] + 61.856;
   1:L PR[91] R[100]mm/sec CNT100;
   1:  PR[91,1] = PR[90,1] + -4.957;
   1:  PR[91,2] = PR[90,2] + 23.942;
   1:  PR[91,3] = PR[90,3] + 61.868;
   1:L PR[91] R[100]mm/sec CNT100;
   1:  PR[91,1] = PR[90,1] + -6.201;
   1:  PR[91,2] = PR[90,2] + 23.694;
   1:  PR[91,3] = PR[90,3] + 61.878;
   1:L PR[91] R[100]mm/sec CNT100;
   1:  PR[91,1] = PR[90,1] + -7.428;
   1:  PR[91,2] = PR[90,2] + 23.381;
   1:  PR[91,3] = PR[90,3] + 61.889;
   1:L PR[91] R[100]mm/sec CNT100;
   1:  PR[91,1] = PR[90,1] + -8.514;
   1:  PR[91,2] = PR[90,2] + 23.045;
   1:  PR[91,3] = PR[90,3] + 61.900;
   1:L PR[91] R[100]mm/sec CNT100;
   1:  PR[91,1] = PR[90,1] + -9.705;
   1:  PR[91,2] = PR[90,2] + 22.610;
   1:  PR[91,3] = PR[90,3] + 61.910;
   1:L PR[91] R[100]mm/sec CNT100;
   1:  PR[91,1] = PR[90,1] + -10.868;
   1:  PR[91,2] = PR[90,2] + 22.115;
   1:  PR[91,3] = PR[90,3] + 61.921;
   1:L PR[91] R[100]mm/sec CNT100;
   1:  PR[91,1] = PR[90,1] + -12.003;
   1:  PR[91,2] = PR[90,2] + 21.560;
   1:  PR[91,3] = PR[90,3] + 61.932;
   1:L PR[91] R[100]mm/sec CNT100;
   1:  PR[91,1] = PR[90,1] + -13.104;
   1:  PR[91,2] = PR[90,2] + 20.947;
   1:  PR[91,3] = PR[90,3] + 61.943;
   1:L PR[91] R[100]mm/sec CNT100;
   1:  PR[91,1] = PR[90,1] + -14.172;
   1:  PR[91,2] = PR[90,2] + 20.278;
   1:  PR[91,3] = PR[90,3] + 61.954;
   1:L PR[91] R[100]mm/sec CNT100;
   1:  PR[91,1] = PR[90,1] + -15.119;
   1:  PR[91,2] = PR[90,2] + 19.615;
   1:  PR[91,3] = PR[90,3] + 61.965;
   1:L PR[91] R[100]mm/sec CNT100;
   1:  PR[91,1] = PR[90,1] + -16.113;
   1:  PR[91,2] = PR[90,2] + 18.842;
   1:  PR[91,3] = PR[90,3] + 61.975;
   1:L PR[91] R[100]mm/sec CNT100;
   1:  PR[91,1] = PR[90,1] + -17.064;
   1:  PR[91,2] = PR[90,2] + 18.019;
   1:  PR[91,3] = PR[90,3] + 61.986;
   1:L PR[91] R[100]mm/sec CNT100;
   1:  PR[91,1] = PR[90,1] + -17.975;
   1:  PR[91,2] = PR[90,2] + 17.142;
   1:  PR[91,3] = PR[90,3] + 61.997;
   1:L PR[91] R[100]mm/sec CNT100;
   1:  PR[91,1] = PR[90,1] + -18.776;
   1:  PR[91,2] = PR[90,2] + 16.288;
   1:  PR[91,3] = PR[90,3] + 62.008;
   1:L PR[91] R[100]mm/sec CNT100;
   1:  PR[91,1] = PR[90,1] + -19.646;
   1:  PR[91,2] = PR[90,2] + 15.257;
   1:  PR[91,3] = PR[90,3] + 62.018;
   1:L PR[91] R[100]mm/sec CNT100;
   1:  PR[91,1] = PR[90,1] + -20.355;
   1:  PR[91,2] = PR[90,2] + 14.321;
   1:  PR[91,3] = PR[90,3] + 62.030;
   1:L PR[91] R[100]mm/sec CNT100;
   1:  PR[91,1] = PR[90,1] + -21.063;
   1:  PR[91,2] = PR[90,2] + 13.280;
   1:  PR[91,3] = PR[90,3] + 62.040;
   1:L PR[91] R[100]mm/sec CNT100;
   1:  PR[91,1] = PR[90,1] + -21.676;
   1:  PR[91,2] = PR[90,2] + 12.272;
   1:  PR[91,3] = PR[90,3] + 62.051;
   1:L PR[91] R[100]mm/sec CNT100;
   1:  PR[91,1] = PR[90,1] + -22.273;
   1:  PR[91,2] = PR[90,2] + 11.166;
   1:  PR[91,3] = PR[90,3] + 62.061;
   1:L PR[91] R[100]mm/sec CNT100;
   1:  PR[91,1] = PR[90,1] + -22.811;
   1:  PR[91,2] = PR[90,2] + 10.031;
   1:  PR[91,3] = PR[90,3] + 62.072;
   1:L PR[91] R[100]mm/sec CNT100;
   1:  PR[91,1] = PR[90,1] + -23.287;
   1:  PR[91,2] = PR[90,2] + 8.872;
   1:  PR[91,3] = PR[90,3] + 62.083;
   1:L PR[91] R[100]mm/sec CNT100;
   1:  PR[91,1] = PR[90,1] + -23.701;
   1:  PR[91,2] = PR[90,2] + 7.690;
   1:  PR[91,3] = PR[90,3] + 62.094;
   1:L PR[91] R[100]mm/sec CNT100;
   1:  PR[91,1] = PR[90,1] + -24.052;
   1:  PR[91,2] = PR[90,2] + 6.489;
   1:  PR[91,3] = PR[90,3] + 62.104;
   1:L PR[91] R[100]mm/sec CNT100;
   1:  PR[91,1] = PR[90,1] + -24.326;
   1:  PR[91,2] = PR[90,2] + 5.335;
   1:  PR[91,3] = PR[90,3] + 62.115;
   1:L PR[91] R[100]mm/sec CNT100;
   1:  PR[91,1] = PR[90,1] + -24.552;
   1:  PR[91,2] = PR[90,2] + 4.104;
   1:  PR[91,3] = PR[90,3] + 62.126;
   1:L PR[91] R[100]mm/sec CNT100;
   1:  PR[91,1] = PR[90,1] + -24.713;
   1:  PR[91,2] = PR[90,2] + 2.864;
   1:  PR[91,3] = PR[90,3] + 62.136;
   1:L PR[91] R[100]mm/sec CNT100;
   1:  PR[91,1] = PR[90,1] + -24.808;
   1:  PR[91,2] = PR[90,2] + 1.617;
   1:  PR[91,3] = PR[90,3] + 62.147;
   1:L PR[91] R[100]mm/sec CNT100;
   1:  PR[91,1] = PR[90,1] + -24.839;
   1:  PR[91,2] = PR[90,2] + 0.428;
   1:  PR[91,3] = PR[90,3] + 62.158;
   1:L PR[91] R[100]mm/sec CNT100;
   1:  PR[91,1] = PR[90,1] + -24.806;
   1:  PR[91,2] = PR[90,2] + -0.823;
   1:  PR[91,3] = PR[90,3] + 62.168;
   1:L PR[91] R[100]mm/sec CNT100;
   1:  PR[91,1] = PR[90,1] + -24.707;
   1:  PR[91,2] = PR[90,2] + -2.070;
   1:  PR[91,3] = PR[90,3] + 62.179;
   1:L PR[91] R[100]mm/sec CNT100;
   1:  PR[91,1] = PR[90,1] + -24.542;
   1:  PR[91,2] = PR[90,2] + -3.311;
   1:  PR[91,3] = PR[90,3] + 62.190;
   1:L PR[91] R[100]mm/sec CNT100;
   1:  PR[91,1] = PR[90,1] + -24.326;
   1:  PR[91,2] = PR[90,2] + -4.479;
   1:  PR[91,3] = PR[90,3] + 62.201;
   1:L PR[91] R[100]mm/sec CNT100;
   1:  PR[91,1] = PR[90,1] + -24.036;
   1:  PR[91,2] = PR[90,2] + -5.696;
   1:  PR[91,3] = PR[90,3] + 62.211;
   1:L PR[91] R[100]mm/sec CNT100;
   1:  PR[91,1] = PR[90,1] + -23.680;
   1:  PR[91,2] = PR[90,2] + -6.898;
   1:  PR[91,3] = PR[90,3] + 62.222;
   1:L PR[91] R[100]mm/sec CNT100;
   1:  PR[91,1] = PR[90,1] + -23.287;
   1:  PR[91,2] = PR[90,2] + -8.016;
   1:  PR[91,3] = PR[90,3] + 62.233;
   1:L PR[91] R[100]mm/sec CNT100;
   1:  PR[91,1] = PR[90,1] + -22.811;
   1:  PR[91,2] = PR[90,2] + -9.176;
   1:  PR[91,3] = PR[90,3] + 62.243;
   1:L PR[91] R[100]mm/sec CNT100;
   1:  PR[91,1] = PR[90,1] + -22.302;
   1:  PR[91,2] = PR[90,2] + -10.254;
   1:  PR[91,3] = PR[90,3] + 62.254;
   1:L PR[91] R[100]mm/sec CNT100;
   1:  PR[91,1] = PR[90,1] + -22.276;
   1:  PR[91,2] = PR[90,2] + -10.306;
   1:  PR[91,3] = PR[90,3] + 62.265;
   1:L PR[91] R[100]mm/sec CNT100;
   1:  PR[91,1] = PR[90,1] + -21.676;
   1:  PR[91,2] = PR[90,2] + -11.417;
   1:L PR[91] R[100]mm/sec CNT100;
   1:  PR[91,1] = PR[90,1] + -21.063;
   1:  PR[91,2] = PR[90,2] + -12.425;
   1:  PR[91,3] = PR[90,3] + 62.276;
   1:L PR[91] R[100]mm/sec CNT100;
   1:  PR[91,1] = PR[90,1] + -20.356;
   1:  PR[91,2] = PR[90,2] + -13.466;
   1:  PR[91,3] = PR[90,3] + 62.286;
   1:L PR[91] R[100]mm/sec CNT100;
   1:  PR[91,1] = PR[90,1] + -19.593;
   1:  PR[91,2] = PR[90,2] + -14.469;
   1:  PR[91,3] = PR[90,3] + 62.297;
   1:L PR[91] R[100]mm/sec CNT100;
   1:  PR[91,1] = PR[90,1] + -18.836;
   1:  PR[91,2] = PR[90,2] + -15.366;
   1:  PR[91,3] = PR[90,3] + 62.308;
   1:L PR[91] R[100]mm/sec CNT100;
   1:  PR[91,1] = PR[90,1] + -17.975;
   1:  PR[91,2] = PR[90,2] + -16.287;
   1:  PR[91,3] = PR[90,3] + 62.318;
   1:L PR[91] R[100]mm/sec CNT100;
   1:  PR[91,1] = PR[90,1] + -17.064;
   1:  PR[91,2] = PR[90,2] + -17.164;
   1:  PR[91,3] = PR[90,3] + 62.329;
   1:L PR[91] R[100]mm/sec CNT100;
   1:  PR[91,1] = PR[90,1] + -16.188;
   1:  PR[91,2] = PR[90,2] + -17.924;
   1:  PR[91,3] = PR[90,3] + 62.340;
   1:L PR[91] R[100]mm/sec CNT100;
   1:  PR[91,1] = PR[90,1] + -15.118;
   1:  PR[91,2] = PR[90,2] + -18.760;
   1:  PR[91,3] = PR[90,3] + 62.350;
   1:L PR[91] R[100]mm/sec CNT100;
   1:  PR[91,1] = PR[90,1] + -14.172;
   1:  PR[91,2] = PR[90,2] + -19.422;
   1:  PR[91,3] = PR[90,3] + 62.362;
   1:L PR[91] R[100]mm/sec CNT100;
   1:  PR[91,1] = PR[90,1] + -13.010;
   1:  PR[91,2] = PR[90,2] + -20.147;
   1:  PR[91,3] = PR[90,3] + 62.372;
   1:L PR[91] R[100]mm/sec CNT100;
   1:  PR[91,1] = PR[90,1] + -12.003;
   1:  PR[91,2] = PR[90,2] + -20.705;
   1:  PR[91,3] = PR[90,3] + 62.384;
   1:L PR[91] R[100]mm/sec CNT100;
   1:  PR[91,1] = PR[90,1] + -10.869;
   1:  PR[91,2] = PR[90,2] + -21.260;
   1:  PR[91,3] = PR[90,3] + 62.394;
   1:L PR[91] R[100]mm/sec CNT100;
   1:  PR[91,1] = PR[90,1] + -9.705;
   1:  PR[91,2] = PR[90,2] + -21.755;
   1:  PR[91,3] = PR[90,3] + 62.405;
   1:L PR[91] R[100]mm/sec CNT100;
   1:  PR[91,1] = PR[90,1] + -8.515;
   1:  PR[91,2] = PR[90,2] + -22.190;
   1:  PR[91,3] = PR[90,3] + 62.416;
   1:L PR[91] R[100]mm/sec CNT100;
   1:  PR[91,1] = PR[90,1] + -7.428;
   1:  PR[91,2] = PR[90,2] + -22.525;
   1:  PR[91,3] = PR[90,3] + 62.427;
   1:L PR[91] R[100]mm/sec CNT100;
   1:  PR[91,1] = PR[90,1] + -6.201;
   1:  PR[91,2] = PR[90,2] + -22.839;
   1:  PR[91,3] = PR[90,3] + 62.437;
   1:L PR[91] R[100]mm/sec CNT100;
   1:  PR[91,1] = PR[90,1] + -4.958;
   1:  PR[91,2] = PR[90,2] + -23.087;
   1:  PR[91,3] = PR[90,3] + 62.448;
   1:L PR[91] R[100]mm/sec CNT100;
   1:  PR[91,1] = PR[90,1] + -3.702;
   1:  PR[91,2] = PR[90,2] + -23.269;
   1:  PR[91,3] = PR[90,3] + 62.459;
   1:L PR[91] R[100]mm/sec CNT100;
   1:  PR[91,1] = PR[90,1] + -2.435;
   1:  PR[91,2] = PR[90,2] + -23.385;
   1:  PR[91,3] = PR[90,3] + 62.470;
   1:L PR[91] R[100]mm/sec CNT100;
   1:  PR[91,1] = PR[90,1] + -1.314;
   1:  PR[91,2] = PR[90,2] + -23.432;
   1:  PR[91,3] = PR[90,3] + 62.481;
   1:L PR[91] R[100]mm/sec CNT100;
   1:  PR[91,1] = PR[90,1] + 0.922;
   1:  PR[91,2] = PR[90,2] + -23.434;
   1:  PR[91,3] = PR[90,3] + 62.491;
   1:L PR[91] R[100]mm/sec CNT100;
   1:  PR[91] = PR[90];
   1:  PR[91,1] = PR[90,1] + 1.623;
   1:  PR[91,2] = PR[90,2] + -23.723;
   1:  PR[91,3] = PR[90,3] + 63.840;
   1:L PR[91] R[100]mm/sec CNT100;
   1:  PR[91,1] = PR[90,1] + 2.962;
   1:  PR[91,2] = PR[90,2] + -23.606;
   1:  PR[91,3] = PR[90,3] + 62.522;
   1:L PR[91] R[100]mm/sec CNT100;
   1:  PR[91,1] = PR[90,1] + 4.290;
   1:  PR[91,2] = PR[90,2] + -23.415;
   1:  PR[91,3] = PR[90,3] + 62.533;
   1:L PR[91] R[100]mm/sec CNT100;
   1:  PR[91,1] = PR[90,1] + 5.608;
   1:  PR[91,2] = PR[90,2] + -23.150;
   1:  PR[91,3] = PR[90,3] + 62.545;
   1:L PR[91] R[100]mm/sec CNT100;
   1:  PR[91,1] = PR[90,1] + 6.440;
   1:  PR[91,2] = PR[90,2] + -22.942;
   1:  PR[91,3] = PR[90,3] + 62.557;
   1:L PR[91] R[100]mm/sec CNT100;
   1:  PR[91,1] = PR[90,1] + 7.729;
   1:  PR[91,2] = PR[90,2] + -22.559;
   1:  PR[91,3] = PR[90,3] + 62.564;
   1:L PR[91] R[100]mm/sec CNT100;
   1:  PR[91,1] = PR[90,1] + 8.992;
   1:  PR[91,2] = PR[90,2] + -22.106;
   1:  PR[91,3] = PR[90,3] + 62.576;
   1:L PR[91] R[100]mm/sec CNT100;
   1:  PR[91,1] = PR[90,1] + 10.229;
   1:  PR[91,2] = PR[90,2] + -21.584;
   1:  PR[91,3] = PR[90,3] + 62.587;
   1:L PR[91] R[100]mm/sec CNT100;
   1:  PR[91,1] = PR[90,1] + 11.012;
   1:  PR[91,2] = PR[90,2] + -21.207;
   1:  PR[91,3] = PR[90,3] + 62.599;
   1:L PR[91] R[100]mm/sec CNT100;
   1:  PR[91,1] = PR[90,1] + 11.426;
   1:  PR[91,2] = PR[90,2] + -20.998;
   1:  PR[91,3] = PR[90,3] + 62.607;
   1:L PR[91] R[100]mm/sec CNT100;
   1:  PR[91,1] = PR[90,1] + 12.598;
   1:  PR[91,2] = PR[90,2] + -20.341;
   1:  PR[91,3] = PR[90,3] + 62.611;
   1:L PR[91] R[100]mm/sec CNT100;
   1:  PR[91,1] = PR[90,1] + 13.728;
   1:  PR[91,2] = PR[90,2] + -19.624;
   1:  PR[91,3] = PR[90,3] + 62.622;
   1:L PR[91] R[100]mm/sec CNT100;
   1:  PR[91,1] = PR[90,1] + 14.818;
   1:  PR[91,2] = PR[90,2] + -18.844;
   1:  PR[91,3] = PR[90,3] + 62.634;
   1:L PR[91] R[100]mm/sec CNT100;
   1:  PR[91,1] = PR[90,1] + 15.500;
   1:  PR[91,2] = PR[90,2] + -18.309;
   1:  PR[91,3] = PR[90,3] + 62.646;
   1:L PR[91] R[100]mm/sec CNT100;
   1:  PR[91,1] = PR[90,1] + 16.515;
   1:  PR[91,2] = PR[90,2] + -17.434;
   1:  PR[91,3] = PR[90,3] + 62.653;
   1:L PR[91] R[100]mm/sec CNT100;
   1:  PR[91,1] = PR[90,1] + 17.506;
   1:  PR[91,2] = PR[90,2] + -16.476;
   1:  PR[91,3] = PR[90,3] + 62.665;
   1:L PR[91] R[100]mm/sec CNT100;
   1:  PR[91,1] = PR[90,1] + 18.442;
   1:  PR[91,2] = PR[90,2] + -15.463;
   1:  PR[91,3] = PR[90,3] + 62.677;
   1:L PR[91] R[100]mm/sec CNT100;
   1:  PR[91,1] = PR[90,1] + 19.016;
   1:  PR[91,2] = PR[90,2] + -14.781;
   1:  PR[91,3] = PR[90,3] + 62.689;
   1:L PR[91] R[100]mm/sec CNT100;
   1:  PR[91,1] = PR[90,1] + 19.853;
   1:  PR[91,2] = PR[90,2] + -13.685;
   1:  PR[91,3] = PR[90,3] + 62.696;
   1:L PR[91] R[100]mm/sec CNT100;
   1:  PR[91,1] = PR[90,1] + 20.625;
   1:  PR[91,2] = PR[90,2] + -12.543;
   1:  PR[91,3] = PR[90,3] + 62.708;
   1:L PR[91] R[100]mm/sec CNT100;
   1:  PR[91,1] = PR[90,1] + 21.090;
   1:  PR[91,2] = PR[90,2] + -11.780;
   1:  PR[91,3] = PR[90,3] + 62.720;
   1:L PR[91] R[100]mm/sec CNT100;
   1:  PR[91,1] = PR[90,1] + 21.753;
   1:  PR[91,2] = PR[90,2] + -10.572;
   1:  PR[91,3] = PR[90,3] + 62.728;
   1:L PR[91] R[100]mm/sec CNT100;
   1:  PR[91,1] = PR[90,1] + 22.344;
   1:  PR[91,2] = PR[90,2] + -9.331;
   1:  PR[91,3] = PR[90,3] + 62.740;
   1:L PR[91] R[100]mm/sec CNT100;
   1:  PR[91,1] = PR[90,1] + 22.864;
   1:  PR[91,2] = PR[90,2] + -8.056;
   1:  PR[91,3] = PR[90,3] + 62.752;
   1:L PR[91] R[100]mm/sec CNT100;
   1:  PR[91,1] = PR[90,1] + 23.162;
   1:  PR[91,2] = PR[90,2] + -7.211;
   1:  PR[91,3] = PR[90,3] + 62.764;
   1:L PR[91] R[100]mm/sec CNT100;
   1:  PR[91,1] = PR[90,1] + 23.562;
   1:  PR[91,2] = PR[90,2] + -5.889;
   1:  PR[91,3] = PR[90,3] + 62.772;
   1:L PR[91] R[100]mm/sec CNT100;
   1:  PR[91,1] = PR[90,1] + 23.678;
   1:  PR[91,2] = PR[90,2] + -5.440;
   1:  PR[91,3] = PR[90,3] + 62.784;
   1:L PR[91] R[100]mm/sec CNT100;
   1:  PR[91,1] = PR[90,1] + 23.882;
   1:  PR[91,2] = PR[90,2] + -4.561;
   1:  PR[91,3] = PR[90,3] + 62.788;
   1:L PR[91] R[100]mm/sec CNT100;
   1:  PR[91,1] = PR[90,1] + 24.128;
   1:  PR[91,2] = PR[90,2] + -3.205;
   1:  PR[91,3] = PR[90,3] + 62.795;
   1:L PR[91] R[100]mm/sec CNT100;
   1:  PR[91,1] = PR[90,1] + 24.246;
   1:  PR[91,2] = PR[90,2] + -2.316;
   1:  PR[91,3] = PR[90,3] + 62.807;
   1:L PR[91] R[100]mm/sec CNT100;
   1:  PR[91,1] = PR[90,1] + 24.364;
   1:  PR[91,2] = PR[90,2] + -0.945;
   1:  PR[91,3] = PR[90,3] + 62.815;
   1:L PR[91] R[100]mm/sec CNT100;
   1:  PR[91,1] = PR[90,1] + 24.403;
   1:  PR[91,2] = PR[90,2] + 0.428;
   1:  PR[91,3] = PR[90,3] + 62.827;
   1:L PR[91] R[100]mm/sec CNT100;
   1:  PR[91,1] = PR[90,1] + 24.364;
   1:  PR[91,2] = PR[90,2] + 1.800;
   1:  PR[91,3] = PR[90,3] + 62.839;
   1:L PR[91] R[100]mm/sec CNT100;
   1:  PR[91,1] = PR[90,1] + 24.246;
   1:  PR[91,2] = PR[90,2] + 3.171;
   1:  PR[91,3] = PR[90,3] + 62.851;
   1:L PR[91] R[100]mm/sec CNT100;
   1:  PR[91,1] = PR[90,1] + 24.128;
   1:  PR[91,2] = PR[90,2] + 4.060;
   1:  PR[91,3] = PR[90,3] + 62.863;
   1:L PR[91] R[100]mm/sec CNT100;
   1:  PR[91,1] = PR[90,1] + 23.883;
   1:  PR[91,2] = PR[90,2] + 5.414;
   1:  PR[91,3] = PR[90,3] + 62.871;
   1:L PR[91] R[100]mm/sec CNT100;
   1:  PR[91,1] = PR[90,1] + 23.561;
   1:  PR[91,2] = PR[90,2] + 6.749;
   1:  PR[91,3] = PR[90,3] + 62.883;
   1:L PR[91] R[100]mm/sec CNT100;
   1:  PR[91,1] = PR[90,1] + 23.162;
   1:  PR[91,2] = PR[90,2] + 8.067;
   1:  PR[91,3] = PR[90,3] + 62.895;
   1:L PR[91] R[100]mm/sec CNT100;
   1:  PR[91,1] = PR[90,1] + 22.864;
   1:  PR[91,2] = PR[90,2] + 8.911;
   1:  PR[91,3] = PR[90,3] + 62.907;
   1:L PR[91] R[100]mm/sec CNT100;
   1:  PR[91,1] = PR[90,1] + 22.343;
   1:  PR[91,2] = PR[90,2] + 10.188;
   1:  PR[91,3] = PR[90,3] + 62.914;
   1:L PR[91] R[100]mm/sec CNT100;
   1:  PR[91,1] = PR[90,1] + 21.963;
   1:  PR[91,2] = PR[90,2] + 11.004;
   1:  PR[91,3] = PR[90,3] + 62.926;
   1:L PR[91] R[100]mm/sec CNT100;
   1:  PR[91,1] = PR[90,1] + 21.754;
   1:  PR[91,2] = PR[90,2] + 11.425;
   1:  PR[91,3] = PR[90,3] + 62.934;
   1:L PR[91] R[100]mm/sec CNT100;
   1:  PR[91,1] = PR[90,1] + 21.330;
   1:  PR[91,2] = PR[90,2] + 12.217;
   1:  PR[91,3] = PR[90,3] + 62.938;
   1:L PR[91] R[100]mm/sec CNT100;
   1:  PR[91,1] = PR[90,1] + 20.622;
   1:  PR[91,2] = PR[90,2] + 13.403;
   1:  PR[91,3] = PR[90,3] + 62.946;
   1:L PR[91] R[100]mm/sec CNT100;
   1:  PR[91,1] = PR[90,1] + 20.127;
   1:  PR[91,2] = PR[90,2] + 14.146;
   1:  PR[91,3] = PR[90,3] + 62.958;
   1:L PR[91] R[100]mm/sec CNT100;
   1:  PR[91,1] = PR[90,1] + 19.567;
   1:  PR[91,2] = PR[90,2] + 14.925;
   1:  PR[91,3] = PR[90,3] + 62.966;
   1:L PR[91] R[100]mm/sec CNT100;
   1:  PR[91,1] = PR[90,1] + 19.019;
   1:  PR[91,2] = PR[90,2] + 15.632;
   1:  PR[91,3] = PR[90,3] + 62.974;
   1:L PR[91] R[100]mm/sec CNT100;
   1:  PR[91,1] = PR[90,1] + 18.118;
   1:  PR[91,2] = PR[90,2] + 16.681;
   1:  PR[91,3] = PR[90,3] + 62.982;
   1:L PR[91] R[100]mm/sec CNT100;
   1:  PR[91,1] = PR[90,1] + 17.508;
   1:  PR[91,2] = PR[90,2] + 17.329;
   1:  PR[91,3] = PR[90,3] + 62.994;
   1:L PR[91] R[100]mm/sec CNT100;
   1:  PR[91,1] = PR[90,1] + 16.515;
   1:  PR[91,2] = PR[90,2] + 18.289;
   1:  PR[91,3] = PR[90,3] + 63.001;
   1:L PR[91] R[100]mm/sec CNT100;
   1:  PR[91,1] = PR[90,1] + 15.502;
   1:  PR[91,2] = PR[90,2] + 19.162;
   1:  PR[91,3] = PR[90,3] + 63.013;
   1:L PR[91] R[100]mm/sec CNT100;
   1:  PR[91,1] = PR[90,1] + 14.440;
   1:  PR[91,2] = PR[90,2] + 19.981;
   1:  PR[91,3] = PR[90,3] + 63.025;
   1:L PR[91] R[100]mm/sec CNT100;
   1:  PR[91,1] = PR[90,1] + 13.730;
   1:  PR[91,2] = PR[90,2] + 20.478;
   1:  PR[91,3] = PR[90,3] + 63.037;
   1:L PR[91] R[100]mm/sec CNT100;
   1:  PR[91,1] = PR[90,1] + 12.598;
   1:  PR[91,2] = PR[90,2] + 21.197;
   1:  PR[91,3] = PR[90,3] + 63.044;
   1:L PR[91] R[100]mm/sec CNT100;
   1:  PR[91,1] = PR[90,1] + 11.430;
   1:  PR[91,2] = PR[90,2] + 21.851;
   1:  PR[91,3] = PR[90,3] + 63.056;
   1:L PR[91] R[100]mm/sec CNT100;
   1:  PR[91,1] = PR[90,1] + 10.226;
   1:  PR[91,2] = PR[90,2] + 22.440;
   1:  PR[91,3] = PR[90,3] + 63.067;
   1:L PR[91] R[100]mm/sec CNT100;
   1:  PR[91,1] = PR[90,1] + 8.989;
   1:  PR[91,2] = PR[90,2] + 22.962;
   1:  PR[91,3] = PR[90,3] + 63.079;
   1:L PR[91] R[100]mm/sec CNT100;
   1:  PR[91,1] = PR[90,1] + 8.183;
   1:  PR[91,2] = PR[90,2] + 23.260;
   1:  PR[91,3] = PR[90,3] + 63.091;
   1:L PR[91] R[100]mm/sec CNT100;
   1:  PR[91,1] = PR[90,1] + 6.903;
   1:  PR[91,2] = PR[90,2] + 23.669;
   1:  PR[91,3] = PR[90,3] + 63.098;
   1:L PR[91] R[100]mm/sec CNT100;
   1:  PR[91,1] = PR[90,1] + 5.605;
   1:  PR[91,2] = PR[90,2] + 24.005;
   1:  PR[91,3] = PR[90,3] + 63.110;
   1:L PR[91] R[100]mm/sec CNT100;
   1:  PR[91,1] = PR[90,1] + 4.287;
   1:  PR[91,2] = PR[90,2] + 24.270;
   1:  PR[91,3] = PR[90,3] + 63.122;
   1:L PR[91] R[100]mm/sec CNT100;
   1:  PR[91,1] = PR[90,1] + 3.444;
   1:  PR[91,2] = PR[90,2] + 24.399;
   1:  PR[91,3] = PR[90,3] + 63.133;
   1:L PR[91] R[100]mm/sec CNT100;
   1:  PR[91,1] = PR[90,1] + 2.106;
   1:  PR[91,2] = PR[90,2] + 24.544;
   1:  PR[91,3] = PR[90,3] + 63.141;
   1:L PR[91] R[100]mm/sec CNT100;
   1:  PR[91,1] = PR[90,1] + 0.764;
   1:  PR[91,2] = PR[90,2] + 24.614;
   1:  PR[91,3] = PR[90,3] + 63.152;
   1:L PR[91] R[100]mm/sec CNT100;
   1:  PR[91,1] = PR[90,1] + -0.515;
   1:  PR[91,2] = PR[90,2] + 24.621;
   1:  PR[91,3] = PR[90,3] + 63.164;
   1:L PR[91] R[100]mm/sec CNT100;
   1:  PR[91,1] = PR[90,1] + -1.865;
   1:  PR[91,2] = PR[90,2] + 24.578;
   1:  PR[91,3] = PR[90,3] + 63.175;
   1:L PR[91] R[100]mm/sec CNT100;
   1:  PR[91,1] = PR[90,1] + -2.719;
   1:  PR[91,2] = PR[90,2] + 24.509;
   1:  PR[91,3] = PR[90,3] + 63.187;
   1:L PR[91] R[100]mm/sec CNT100;
   1:  PR[91,1] = PR[90,1] + -3.681;
   1:  PR[91,2] = PR[90,2] + 24.399;
   1:  PR[91,3] = PR[90,3] + 63.194;
   1:L PR[91] R[100]mm/sec CNT100;
   1:  PR[91,1] = PR[90,1] + -4.527;
   1:  PR[91,2] = PR[90,2] + 24.270;
   1:  PR[91,3] = PR[90,3] + 63.203;
   1:L PR[91] R[100]mm/sec CNT100;
   1:  PR[91,1] = PR[90,1] + -5.845;
   1:  PR[91,2] = PR[90,2] + 24.005;
   1:  PR[91,3] = PR[90,3] + 63.210;
   1:L PR[91] R[100]mm/sec CNT100;
   1:  PR[91,1] = PR[90,1] + -7.145;
   1:  PR[91,2] = PR[90,2] + 23.668;
   1:  PR[91,3] = PR[90,3] + 63.222;
   1:L PR[91] R[100]mm/sec CNT100;
   1:  PR[91,1] = PR[90,1] + -7.965;
   1:  PR[91,2] = PR[90,2] + 23.415;
   1:  PR[91,3] = PR[90,3] + 63.233;
   1:L PR[91] R[100]mm/sec CNT100;
   1:  PR[91,1] = PR[90,1] + -9.230;
   1:  PR[91,2] = PR[90,2] + 22.961;
   1:  PR[91,3] = PR[90,3] + 63.241;
   1:L PR[91] R[100]mm/sec CNT100;
   1:  PR[91,1] = PR[90,1] + -10.465;
   1:  PR[91,2] = PR[90,2] + 22.439;
   1:  PR[91,3] = PR[90,3] + 63.252;
   1:L PR[91] R[100]mm/sec CNT100;
   1:  PR[91,1] = PR[90,1] + -11.668;
   1:  PR[91,2] = PR[90,2] + 21.851;
   1:  PR[91,3] = PR[90,3] + 63.264;
   1:L PR[91] R[100]mm/sec CNT100;
   1:  PR[91,1] = PR[90,1] + -12.837;
   1:  PR[91,2] = PR[90,2] + 21.197;
   1:  PR[91,3] = PR[90,3] + 63.276;
   1:L PR[91] R[100]mm/sec CNT100;
   1:  PR[91,1] = PR[90,1] + -13.969;
   1:  PR[91,2] = PR[90,2] + 20.478;
   1:  PR[91,3] = PR[90,3] + 63.287;
   1:L PR[91] R[100]mm/sec CNT100;
   1:  PR[91,1] = PR[90,1] + -14.678;
   1:  PR[91,2] = PR[90,2] + 19.981;
   1:  PR[91,3] = PR[90,3] + 63.299;
   1:L PR[91] R[100]mm/sec CNT100;
   1:  PR[91,1] = PR[90,1] + -15.740;
   1:  PR[91,2] = PR[90,2] + 19.163;
   1:  PR[91,3] = PR[90,3] + 63.306;
   1:L PR[91] R[100]mm/sec CNT100;
   1:  PR[91,1] = PR[90,1] + -16.753;
   1:  PR[91,2] = PR[90,2] + 18.289;
   1:  PR[91,3] = PR[90,3] + 63.318;
   1:L PR[91] R[100]mm/sec CNT100;
   1:  PR[91,1] = PR[90,1] + -17.746;
   1:  PR[91,2] = PR[90,2] + 17.330;
   1:  PR[91,3] = PR[90,3] + 63.330;
   1:L PR[91] R[100]mm/sec CNT100;
   1:  PR[91,1] = PR[90,1] + -18.356;
   1:  PR[91,2] = PR[90,2] + 16.682;
   1:  PR[91,3] = PR[90,3] + 63.342;
   1:L PR[91] R[100]mm/sec CNT100;
   1:  PR[91,1] = PR[90,1] + -19.258;
   1:  PR[91,2] = PR[90,2] + 15.630;
   1:  PR[91,3] = PR[90,3] + 63.349;
   1:L PR[91] R[100]mm/sec CNT100;
   1:  PR[91,1] = PR[90,1] + -19.551;
   1:  PR[91,2] = PR[90,2] + 15.260;
   1:  PR[91,3] = PR[90,3] + 63.361;
   1:L PR[91] R[100]mm/sec CNT100;
   1:  PR[91,1] = PR[90,1] + -20.089;
   1:  PR[91,2] = PR[90,2] + 14.542;
   1:  PR[91,3] = PR[90,3] + 63.366;
   1:L PR[91] R[100]mm/sec CNT100;
   1:  PR[91,1] = PR[90,1] + -20.864;
   1:  PR[91,2] = PR[90,2] + 13.399;
   1:  PR[91,3] = PR[90,3] + 63.373;
   1:L PR[91] R[100]mm/sec CNT100;
   1:  PR[91,1] = PR[90,1] + -21.329;
   1:  PR[91,2] = PR[90,2] + 12.636;
   1:  PR[91,3] = PR[90,3] + 63.385;
   1:L PR[91] R[100]mm/sec CNT100;
   1:  PR[91,1] = PR[90,1] + -21.991;
   1:  PR[91,2] = PR[90,2] + 11.427;
   1:  PR[91,3] = PR[90,3] + 63.393;
   1:L PR[91] R[100]mm/sec CNT100;
   1:  PR[91,1] = PR[90,1] + -22.582;
   1:  PR[91,2] = PR[90,2] + 10.186;
   1:  PR[91,3] = PR[90,3] + 63.405;
   1:L PR[91] R[100]mm/sec CNT100;
   1:  PR[91,1] = PR[90,1] + -23.102;
   1:  PR[91,2] = PR[90,2] + 8.911;
   1:  PR[91,3] = PR[90,3] + 63.417;
   1:L PR[91] R[100]mm/sec CNT100;
   1:  PR[91,1] = PR[90,1] + -23.401;
   1:  PR[91,2] = PR[90,2] + 8.067;
   1:  PR[91,3] = PR[90,3] + 63.429;
   1:L PR[91] R[100]mm/sec CNT100;
   1:  PR[91,1] = PR[90,1] + -23.799;
   1:  PR[91,2] = PR[90,2] + 6.749;
   1:  PR[91,3] = PR[90,3] + 63.437;
   1:L PR[91] R[100]mm/sec CNT100;
   1:  PR[91,1] = PR[90,1] + -24.121;
   1:  PR[91,2] = PR[90,2] + 5.414;
   1:  PR[91,3] = PR[90,3] + 63.449;
   1:L PR[91] R[100]mm/sec CNT100;
   1:  PR[91,1] = PR[90,1] + -24.367;
   1:  PR[91,2] = PR[90,2] + 4.060;
   1:  PR[91,3] = PR[90,3] + 63.461;
   1:L PR[91] R[100]mm/sec CNT100;
   1:  PR[91,1] = PR[90,1] + -24.485;
   1:  PR[91,2] = PR[90,2] + 3.171;
   1:  PR[91,3] = PR[90,3] + 63.472;
   1:L PR[91] R[100]mm/sec CNT100;
   1:  PR[91,1] = PR[90,1] + -24.602;
   1:  PR[91,2] = PR[90,2] + 1.800;
   1:  PR[91,3] = PR[90,3] + 63.480;
   1:L PR[91] R[100]mm/sec CNT100;
   1:  PR[91,1] = PR[90,1] + -24.641;
   1:  PR[91,2] = PR[90,2] + 0.428;
   1:  PR[91,3] = PR[90,3] + 63.492;
   1:L PR[91] R[100]mm/sec CNT100;
   1:  PR[91,1] = PR[90,1] + -24.602;
   1:  PR[91,2] = PR[90,2] + -0.945;
   1:  PR[91,3] = PR[90,3] + 63.504;
   1:L PR[91] R[100]mm/sec CNT100;
   1:  PR[91,1] = PR[90,1] + -24.485;
   1:  PR[91,2] = PR[90,2] + -2.316;
   1:  PR[91,3] = PR[90,3] + 63.516;
   1:L PR[91] R[100]mm/sec CNT100;
   1:  PR[91,1] = PR[90,1] + -24.367;
   1:  PR[91,2] = PR[90,2] + -3.205;
   1:  PR[91,3] = PR[90,3] + 63.528;
   1:L PR[91] R[100]mm/sec CNT100;
   1:  PR[91,1] = PR[90,1] + -24.121;
   1:  PR[91,2] = PR[90,2] + -4.559;
   1:  PR[91,3] = PR[90,3] + 63.536;
   1:L PR[91] R[100]mm/sec CNT100;
   1:  PR[91,1] = PR[90,1] + -23.799;
   1:  PR[91,2] = PR[90,2] + -5.894;
   1:  PR[91,3] = PR[90,3] + 63.548;
   1:L PR[91] R[100]mm/sec CNT100;
   1:  PR[91,1] = PR[90,1] + -23.401;
   1:  PR[91,2] = PR[90,2] + -7.212;
   1:  PR[91,3] = PR[90,3] + 63.560;
   1:L PR[91] R[100]mm/sec CNT100;
   1:  PR[91,1] = PR[90,1] + -23.102;
   1:  PR[91,2] = PR[90,2] + -8.056;
   1:  PR[91,3] = PR[90,3] + 63.572;
   1:L PR[91] R[100]mm/sec CNT100;
   1:  PR[91,1] = PR[90,1] + -22.581;
   1:  PR[91,2] = PR[90,2] + -9.333;
   1:  PR[91,3] = PR[90,3] + 63.579;
   1:L PR[91] R[100]mm/sec CNT100;
   1:  PR[91,1] = PR[90,1] + -22.201;
   1:  PR[91,2] = PR[90,2] + -10.149;
   1:  PR[91,3] = PR[90,3] + 63.591;
   1:L PR[91] R[100]mm/sec CNT100;
   1:  PR[91,1] = PR[90,1] + -21.994;
   1:  PR[91,2] = PR[90,2] + -10.568;
   1:  PR[91,3] = PR[90,3] + 63.599;
   1:L PR[91] R[100]mm/sec CNT100;
   1:  PR[91,1] = PR[90,1] + -21.329;
   1:  PR[91,2] = PR[90,2] + -11.781;
   1:  PR[91,3] = PR[90,3] + 63.603;
   1:L PR[91] R[100]mm/sec CNT100;
   1:  PR[91,1] = PR[90,1] + -20.864;
   1:  PR[91,2] = PR[90,2] + -12.543;
   1:  PR[91,3] = PR[90,3] + 63.615;
   1:L PR[91] R[100]mm/sec CNT100;
   1:  PR[91,1] = PR[90,1] + -20.091;
   1:  PR[91,2] = PR[90,2] + -13.685;
   1:  PR[91,3] = PR[90,3] + 63.623;
   1:L PR[91] R[100]mm/sec CNT100;
   1:  PR[91,1] = PR[90,1] + -19.254;
   1:  PR[91,2] = PR[90,2] + -14.781;
   1:  PR[91,3] = PR[90,3] + 63.635;
   1:L PR[91] R[100]mm/sec CNT100;
   1:  PR[91,1] = PR[90,1] + -18.680;
   1:  PR[91,2] = PR[90,2] + -15.463;
   1:  PR[91,3] = PR[90,3] + 63.647;
   1:L PR[91] R[100]mm/sec CNT100;
   1:  PR[91,1] = PR[90,1] + -17.744;
   1:  PR[91,2] = PR[90,2] + -16.477;
   1:  PR[91,3] = PR[90,3] + 63.655;
   1:L PR[91] R[100]mm/sec CNT100;
   1:  PR[91,1] = PR[90,1] + -16.751;
   1:  PR[91,2] = PR[90,2] + -17.436;
   1:  PR[91,3] = PR[90,3] + 63.667;
   1:L PR[91] R[100]mm/sec CNT100;
   1:  PR[91,1] = PR[90,1] + -16.095;
   1:  PR[91,2] = PR[90,2] + -18.011;
   1:  PR[91,3] = PR[90,3] + 63.678;
   1:L PR[91] R[100]mm/sec CNT100;
   1:  PR[91,1] = PR[90,1] + -15.744;
   1:  PR[91,2] = PR[90,2] + -18.305;
   1:  PR[91,3] = PR[90,3] + 63.686;
   1:L PR[91] R[100]mm/sec CNT100;
   1:  PR[91,1] = PR[90,1] + -14.680;
   1:  PR[91,2] = PR[90,2] + -19.124;
   1:  PR[91,3] = PR[90,3] + 63.690;
   1:L PR[91] R[100]mm/sec CNT100;
   1:  PR[91,1] = PR[90,1] + -13.576;
   1:  PR[91,2] = PR[90,2] + -19.882;
   1:  PR[91,3] = PR[90,3] + 63.702;
   1:L PR[91] R[100]mm/sec CNT100;
   1:  PR[91,1] = PR[90,1] + -12.428;
   1:  PR[91,2] = PR[90,2] + -20.579;
   1:  PR[91,3] = PR[90,3] + 63.713;
   1:L PR[91] R[100]mm/sec CNT100;
   1:  PR[91,1] = PR[90,1] + -11.671;
   1:  PR[91,2] = PR[90,2] + -20.994;
   1:  PR[91,3] = PR[90,3] + 63.725;
   1:L PR[91] R[100]mm/sec CNT100;
   1:  PR[91,1] = PR[90,1] + -10.465;
   1:  PR[91,2] = PR[90,2] + -21.584;
   1:  PR[91,3] = PR[90,3] + 63.732;
   1:L PR[91] R[100]mm/sec CNT100;
   1:  PR[91,1] = PR[90,1] + -9.231;
   1:  PR[91,2] = PR[90,2] + -22.106;
   1:  PR[91,3] = PR[90,3] + 63.744;
   1:L PR[91] R[100]mm/sec CNT100;
   1:  PR[91,1] = PR[90,1] + -7.965;
   1:  PR[91,2] = PR[90,2] + -22.560;
   1:  PR[91,3] = PR[90,3] + 63.756;
   1:L PR[91] R[100]mm/sec CNT100;
   1:  PR[91,1] = PR[90,1] + -7.145;
   1:  PR[91,2] = PR[90,2] + -22.813;
   1:  PR[91,3] = PR[90,3] + 63.767;
   1:L PR[91] R[100]mm/sec CNT100;
   1:  PR[91,1] = PR[90,1] + -5.845;
   1:  PR[91,2] = PR[90,2] + -23.150;
   1:  PR[91,3] = PR[90,3] + 63.775;
   1:L PR[91] R[100]mm/sec CNT100;
   1:  PR[91,1] = PR[90,1] + -4.530;
   1:  PR[91,2] = PR[90,2] + -23.414;
   1:  PR[91,3] = PR[90,3] + 63.787;
   1:L PR[91] R[100]mm/sec CNT100;
   1:  PR[91,1] = PR[90,1] + -3.201;
   1:  PR[91,2] = PR[90,2] + -23.606;
   1:  PR[91,3] = PR[90,3] + 63.798;
   1:L PR[91] R[100]mm/sec CNT100;
   1:  PR[91,1] = PR[90,1] + -1.860;
   1:  PR[91,2] = PR[90,2] + -23.723;
   1:  PR[91,3] = PR[90,3] + 63.810;
   1:L PR[91] R[100]mm/sec CNT100;
   1:  PR[91,1] = PR[90,1] + -1.007;
   1:  PR[91,2] = PR[90,2] + -23.759;
   1:  PR[91,3] = PR[90,3] + 63.821;
   1:L PR[91] R[100]mm/sec CNT100;
   1:  PR[91,1] = PR[90,1] + 0.275;
   1:  PR[91,2] = PR[90,2] + -23.766;
   1:  PR[91,3] = PR[90,3] + 63.829;
   1:L PR[91] R[100]mm/sec CNT100;
   1:  PR[91] = PR[90];
   1:  PR[91,1] = PR[90,1] + 1.280;
   1:  PR[91,2] = PR[90,2] + -23.932;
   1:  PR[91,3] = PR[90,3] + 65.170;
   1:L PR[91] R[100]mm/sec CNT100;
   1:  PR[91,1] = PR[90,1] + 1.945;
   1:  PR[91,2] = PR[90,2] + -23.885;
   1:  PR[91,3] = PR[90,3] + 63.852;
   1:L PR[91] R[100]mm/sec CNT100;
   1:  PR[91,1] = PR[90,1] + 3.290;
   1:  PR[91,2] = PR[90,2] + -23.732;
   1:  PR[91,3] = PR[90,3] + 63.858;
   1:L PR[91] R[100]mm/sec CNT100;
   1:  PR[91,1] = PR[90,1] + 4.050;
   1:  PR[91,2] = PR[90,2] + -23.613;
   1:  PR[91,3] = PR[90,3] + 63.870;
   1:L PR[91] R[100]mm/sec CNT100;
   1:  PR[91,1] = PR[90,1] + 4.710;
   1:  PR[91,2] = PR[90,2] + -23.490;
   1:  PR[91,3] = PR[90,3] + 63.876;
   1:L PR[91] R[100]mm/sec CNT100;
   1:  PR[91,1] = PR[90,1] + 6.027;
   1:  PR[91,2] = PR[90,2] + -23.185;
   1:  PR[91,3] = PR[90,3] + 63.882;
   1:L PR[91] R[100]mm/sec CNT100;
   1:  PR[91,1] = PR[90,1] + 6.765;
   1:  PR[91,2] = PR[90,2] + -22.981;
   1:  PR[91,3] = PR[90,3] + 63.894;
   1:L PR[91] R[100]mm/sec CNT100;
   1:  PR[91,1] = PR[90,1] + 8.017;
   1:  PR[91,2] = PR[90,2] + -22.575;
   1:  PR[91,3] = PR[90,3] + 63.901;
   1:L PR[91] R[100]mm/sec CNT100;
   1:  PR[91,1] = PR[90,1] + 8.680;
   1:  PR[91,2] = PR[90,2] + -22.330;
   1:  PR[91,3] = PR[90,3] + 63.912;
   1:L PR[91] R[100]mm/sec CNT100;
   1:  PR[91,1] = PR[90,1] + 9.258;
   1:  PR[91,2] = PR[90,2] + -22.097;
   1:  PR[91,3] = PR[90,3] + 63.918;
   1:L PR[91] R[100]mm/sec CNT100;
   1:  PR[91,1] = PR[90,1] + 9.969;
   1:  PR[91,2] = PR[90,2] + -21.789;
   1:  PR[91,3] = PR[90,3] + 63.924;
   1:L PR[91] R[100]mm/sec CNT100;
   1:  PR[91,1] = PR[90,1] + 10.609;
   1:  PR[91,2] = PR[90,2] + -21.487;
   1:  PR[91,3] = PR[90,3] + 63.930;
   1:L PR[91] R[100]mm/sec CNT100;
   1:  PR[91,1] = PR[90,1] + 11.218;
   1:  PR[91,2] = PR[90,2] + -21.178;
   1:  PR[91,3] = PR[90,3] + 63.936;
   1:L PR[91] R[100]mm/sec CNT100;
   1:  PR[91,1] = PR[90,1] + 12.443;
   1:  PR[91,2] = PR[90,2] + -20.490;
   1:  PR[91,3] = PR[90,3] + 63.942;
   1:L PR[91] R[100]mm/sec CNT100;
   1:  PR[91,1] = PR[90,1] + 13.076;
   1:  PR[91,2] = PR[90,2] + -20.096;
   1:  PR[91,3] = PR[90,3] + 63.955;
   1:L PR[91] R[100]mm/sec CNT100;
   1:  PR[91,1] = PR[90,1] + 14.129;
   1:  PR[91,2] = PR[90,2] + -19.379;
   1:  PR[91,3] = PR[90,3] + 63.961;
   1:L PR[91] R[100]mm/sec CNT100;
   1:  PR[91,1] = PR[90,1] + 14.747;
   1:  PR[91,2] = PR[90,2] + -18.920;
   1:  PR[91,3] = PR[90,3] + 63.972;
   1:L PR[91] R[100]mm/sec CNT100;
   1:  PR[91,1] = PR[90,1] + 15.235;
   1:  PR[91,2] = PR[90,2] + -18.535;
   1:  PR[91,3] = PR[90,3] + 63.979;
   1:L PR[91] R[100]mm/sec CNT100;
   1:  PR[91,1] = PR[90,1] + 15.830;
   1:  PR[91,2] = PR[90,2] + -18.038;
   1:  PR[91,3] = PR[90,3] + 63.984;
   1:L PR[91] R[100]mm/sec CNT100;
   1:  PR[91,1] = PR[90,1] + 16.296;
   1:  PR[91,2] = PR[90,2] + -17.625;
   1:  PR[91,3] = PR[90,3] + 63.991;
   1:L PR[91] R[100]mm/sec CNT100;
   1:  PR[91,1] = PR[90,1] + 16.817;
   1:  PR[91,2] = PR[90,2] + -17.137;
   1:  PR[91,3] = PR[90,3] + 63.996;
   1:L PR[91] R[100]mm/sec CNT100;
   1:  PR[91,1] = PR[90,1] + 17.340;
   1:  PR[91,2] = PR[90,2] + -16.617;
   1:  PR[91,3] = PR[90,3] + 64.002;
   1:L PR[91] R[100]mm/sec CNT100;
   1:  PR[91,1] = PR[90,1] + 17.890;
   1:  PR[91,2] = PR[90,2] + -16.035;
   1:  PR[91,3] = PR[90,3] + 64.009;
   1:L PR[91] R[100]mm/sec CNT100;
   1:  PR[91,1] = PR[90,1] + 18.322;
   1:  PR[91,2] = PR[90,2] + -15.550;
   1:  PR[91,3] = PR[90,3] + 64.016;
   1:L PR[91] R[100]mm/sec CNT100;
   1:  PR[91,1] = PR[90,1] + 18.834;
   1:  PR[91,2] = PR[90,2] + -14.938;
   1:  PR[91,3] = PR[90,3] + 64.021;
   1:L PR[91] R[100]mm/sec CNT100;
   1:  PR[91,1] = PR[90,1] + 19.667;
   1:  PR[91,2] = PR[90,2] + -13.850;
   1:  PR[91,3] = PR[90,3] + 64.028;
   1:L PR[91] R[100]mm/sec CNT100;
   1:  PR[91,1] = PR[90,1] + 20.088;
   1:  PR[91,2] = PR[90,2] + -13.248;
   1:  PR[91,3] = PR[90,3] + 64.040;
   1:L PR[91] R[100]mm/sec CNT100;
   1:  PR[91,1] = PR[90,1] + 20.526;
   1:  PR[91,2] = PR[90,2] + -12.576;
   1:  PR[91,3] = PR[90,3] + 64.047;
   1:L PR[91] R[100]mm/sec CNT100;
   1:  PR[91,1] = PR[90,1] + 20.865;
   1:  PR[91,2] = PR[90,2] + -12.022;
   1:  PR[91,3] = PR[90,3] + 64.054;
   1:L PR[91] R[100]mm/sec CNT100;
   1:  PR[91,1] = PR[90,1] + 21.263;
   1:  PR[91,2] = PR[90,2] + -11.326;
   1:  PR[91,3] = PR[90,3] + 64.059;
   1:L PR[91] R[100]mm/sec CNT100;
   1:  PR[91,1] = PR[90,1] + 21.569;
   1:  PR[91,2] = PR[90,2] + -10.752;
   1:  PR[91,3] = PR[90,3] + 64.066;
   1:L PR[91] R[100]mm/sec CNT100;
   1:  PR[91,1] = PR[90,1] + 21.924;
   1:  PR[91,2] = PR[90,2] + -10.034;
   1:  PR[91,3] = PR[90,3] + 64.072;
   1:L PR[91] R[100]mm/sec CNT100;
   1:  PR[91,1] = PR[90,1] + 22.195;
   1:  PR[91,2] = PR[90,2] + -9.443;
